	1201:
		_station.arrInfo[E_Language.Chinese]:="Z模组至取Uc位";
		IF M_ZTakeUc() THEN
			_station.iStepNext:=1301;
		END_IF
	1301:
		_station.arrInfo[E_Language.Chinese]:="夹紧气缸夹紧";
		IF G_arrFbCylinder[E_Cylinder.TakeUc1Clamp].M_WorkRequest() THEN
			_station.iStepNext:=1401;
		END_IF
	1401:
		_station.arrInfo[E_Language.Chinese]:="Z模组上升";
		IF M_ZHome() THEN
			_station.iStepNext:=1451;
		END_IF
	1451:
		_station.arrInfo[E_Language.Chinese]:="Y气缸至后位";
		G_arrFbCylinder[E_Cylinder.TakeUc1Y].M_WorkRequest();
		 _station.iStepNext:=1471;
	1471:
		_station.arrInfo[E_Language.Chinese]:="等待气缸到达安全点";
		IF GVL.I.bTakeUc1Y_Cyl_Safe OR GVL.I.bTakeUc1Y_Cyl_W THEN		
			_station.iStepNext:=1501;
		END_IF
	1501:
		_station.arrInfo[E_Language.Chinese]:="等待复位取Uc请求2";
		IF E_MachineType._311 = GVL_Data.stRecipe.eMachineType THEN
			IF NOT  GVL.stHandshake.bTakeUcToTakeUc_M_2 THEN
				GVL.stHandshake.bTakeUc_MToTakeUc_2:=FALSE;
				_station.iStepNext:=1601;
			END_IF
		ELSE
			IF NOT  GVL.stHandshake.bTakeUcToTakeUc_M THEN		
			  GVL.stHandshake.bTakeUc_MToTakeUc:=FALSE;			
				_station.iStepNext:=1551;
			END_IF	 
		END_IF 
	1551:
		_station.arrInfo[E_Language.Chinese]:="旋转气缸旋转";
		IF G_arrFbCylinder[E_Cylinder.TakeUc1Rotate].M_WorkRequest() AND G_arrFbCylinder[E_Cylinder.TakeUc1Y].M_WorkRequest() THEN
			_station.iStepNext:=1601;
		END_IF
	1601:
		_station.arrInfo[E_Language.Chinese]:="向下Uc皮带请求放料";
		GVL.stHandshake.bTakeUc_MToUnloadUcConveyor:=TRUE;
		IF GVL.stHandshake.bUnloadUcConveyorToTakeUc_M THEN
			_station.iStepNext:=1701;
		END_IF
	1701:
		_station.arrInfo[E_Language.Chinese]:="Z气缸下降放Uc";
		IF M_ZPlaceUc() THEN
			_station.iStepNext:=1801;
		END_IF
	1801:
		_station.arrInfo[E_Language.Chinese]:="夹紧气缸松开";
		IF G_arrFbCylinder[E_Cylinder.TakeUc1Clamp].M_HomeRequest() THEN
			_station.iStepNext:=1901;
		END_IF
	1901:
		_station.arrInfo[E_Language.Chinese]:="气缸上升";
		IF M_ZHome() THEN
			_station.iStepNext:=2001;
		END_IF
	2001:
	    _station.arrInfo[E_Language.Chinese]:="复位放料请求";
		GVL.stHandshake.bTakeUc_MToUnloadUcConveyor:=FALSE;
		IF NOT GVL.stHandshake.bUnloadUcConveyorToTakeUc_M THEN
		   	_station.iStepNext:=2101;
		END_IF
	2101:
		_station.arrInfo[E_Language.Chinese]:="旋转气缸复位";
		IF G_arrFbCylinder[E_Cylinder.TakeUc1Rotate].M_HomeRequest() THEN
			_station.iStepNext:=1101;
		END_IF
END_CASE
END_ACTION

ACTION A_Home:
CASE _station.iStepNow OF
	0:
		_station.arrInfo[E_Language.Chinese]:="等待初始化";
		_station.iStepNext:=SEL(_bEnable,1000,100);
	100:
		_station.arrInfo[E_Language.Chinese]:="夹紧气缸松开";
		IF G_arrFbCylinder[E_Cylinder.TakeUc1Clamp].M_HomeRequest() THEN
			_station.iStepNext:=200;
		END_IF
	200:
		_station.arrInfo[E_Language.Chinese]:="Z模组至待料位";
		IF M_ZHome() THEN
			_station.iStepNext:=300;
		END_IF		
	300:
		_station.arrInfo[E_Language.Chinese]:="旋转气缸复位";
		IF G_arrFbCylinder[E_Cylinder.TakeUc1Rotate].M_HomeRequest() THEN
			_station.iStepNext:=400;
		END_IF
	400:
		_station.arrInfo[E_Language.Chinese]:="Y气缸至后位";
	    IF G_arrFbCylinder[E_Cylinder.TakeUc1Y].M_WorkRequest() THEN
		    _station.iStepNext:=1000;
		END_IF
END_CASE
END_ACTION

METHOD M_ZHome : BOOL
VAR_INPUT
END_VAR
CASE GVL_Data.stRecipe.eMachineType OF
	E_MachineType._373:
	M_ZHome:=G_arrFbCylinder[E_Cylinder.TakeUc1Z1].M_HomeRequest();		
	ELSE
	M_ZHome:=G_arrFbCylinder[E_Cylinder.TakeUc1Z1].M_HomeRequest() AND G_arrFbCylinder[E_Cylinder.TakeUc1Z2].M_HomeRequest();
END_CASE
END_METHOD

METHOD M_ZPlaceUc : BOOL
VAR_INPUT
END_VAR
CASE GVL_Data.stRecipe.eMachineType OF
	E_MachineType._373:
	        M_ZPlaceUc:=G_arrFbCylinder[E_Cylinder.TakeUc1Z1].M_WorkRequest();
	E_MachineType._069: 
		    M_ZPlaceUc:=G_arrFbCylinder[E_Cylinder.TakeUc1Z1].M_WorkRequest() AND G_arrFbCylinder[E_Cylinder.TakeUc1Z2].M_WorkRequest();	
    E_MachineType._311:
			M_ZPlaceUc:=G_arrFbCylinder[E_Cylinder.TakeUc1Z1].M_WorkRequest();
	E_MachineType._367:
			M_ZPlaceUc:=G_arrFbCylinder[E_Cylinder.TakeUc1Z1].M_WorkRequest() AND G_arrFbCylinder[E_Cylinder.TakeUc1Z2].M_WorkRequest();
	E_MachineType._200:
	        M_ZPlaceUc:=G_arrFbCylinder[E_Cylinder.TakeUc1Z1].M_WorkRequest() AND G_arrFbCylinder[E_Cylinder.TakeUc1Z2].M_WorkRequest();
END_CASE
END_METHOD

METHOD M_ZTakeUc : BOOL
VAR_INPUT
END_VAR
CASE GVL_Data.stRecipe.eMachineType OF
	E_MachineType._373:
	    M_ZTakeUc:=G_arrFbCylinder[E_Cylinder.TakeUc1Z1].M_WorkRequest();	
	E_MachineType._069:
		    M_ZTakeUc:=G_arrFbCylinder[E_Cylinder.TakeUc1Z1].M_WorkRequest();
	E_MachineType._311:
	    M_ZTakeUc:=G_arrFbCylinder[E_Cylinder.TakeUc1Z1].M_WorkRequest() AND G_arrFbCylinder[E_Cylinder.TakeUc1Z2].M_WorkRequest();
	E_MachineType._367:
			M_ZTakeUc:=G_arrFbCylinder[E_Cylinder.TakeUc1Z2].M_WorkRequest();
	E_MachineType._200:
		   M_ZTakeUc:=G_arrFbCylinder[E_Cylinder.TakeUc1Z1].M_WorkRequest() AND G_arrFbCylinder[E_Cylinder.TakeUc1Z2].M_WorkRequest();
END_CASE
END_METHOD

END_PROGRAM

// ---- POUs/P_StationUnloadFrock.TcPOU
PROGRAM P_StationUnloadFrock
VAR
	_station:					REFERENCE TO ST_SystemStation;
	_bEnable: 					BOOL;
	
	_UnloadFrockCheck0FTrig:         Tc2_Standard.F_TRIG;
	
END_VAR

_station REF= G_arrStation[E_Station.UnloadFrock];
_station.arrName[E_Language.Chinese]:="下工装";
_station.arrName[E_Language.Vietnamese]:="Công cụ tiếp theo";
_bEnable:=NOT GVL.stSetting.arrStationShield[E_Station.UnloadFrock];
A_Auto();
A_Home();

_UnloadFrockCheck0FTrig(CLK:= GVL.I.bUnloadFrockCheck0, Q=> );

ACTION A_Auto:
CASE _station.iStepNow OF
	1000:
		_station.arrInfo[E_Language.Chinese]:="初始化完成等待启动";
		IF _bEnable THEN
			_station.iStepNext:=1101;
		END_IF
	1101:
		_station.arrInfo[E_Language.Chinese]:="判断是否有料";
		IF NOT GVL.I.bUnloadFrockCheck1 THEN
			_station.iStepNext:=1201;
		END_IF
	1201:
		_station.arrInfo[E_Language.Chinese]:="请求取Uc站放料";
		 GVL.stHandshake.bUnloadFrockToTakeUc:=TRUE;
		 IF  GVL.stHandshake.bTakeUcToUnloadFrock THEN
			 _station.iStepNext:=1301;
		 END_IF
	1301://安装了下工装站流入传感器但未移至阻挡气缸后侧启用此条
		_station.arrInfo[E_Language.Chinese]:="等待产品流入";
		GVL.stOverTime.bUnloadFrockCheck1:=TRUE; 
		IF NOT GVL.I.bTakeUcCheck1 AND GVL.I.bUnloadFrockCheck0 THEN
			GVL.stOverTime.bUnloadFrockCheck1:=FALSE; 
			_station.iStepNext:=1401;
		END_IF
		
(*	1301://安装了下工装站流入传感器并且移到了阻挡气缸后侧启用此条
		_station.arrInfo[E_Language.Chinese]:="等待产品从取UC站流出";
		GVL.stOverTime.bUnloadFrockCheck1:=TRUE; 
		IF NOT GVL.I.bTakeUcCheck1 THEN
			GVL.stOverTime.bUnloadFrockCheck1:=FALSE; 
			_station.iStepNext:=1311;
		END_IF		
	1311:		
		_station.arrInfo[E_Language.Chinese]:="产品从取UC站流出确认";
		IF _UnloadFrockCheck0FTrig.Q THEN
			_station.iStepNext:=1401;
		END_IF	*)	
	
	1401:
		_station.arrInfo[E_Language.Chinese]:="复位请求信号";
		 GVL.stHandshake.bUnloadFrockToTakeUc:=FALSE;
		 IF NOT GVL.stHandshake.bTakeUcToUnloadFrock THEN
			 _station.iStepNext:=1501;
		 END_IF
	1501:
		_station.arrInfo[E_Language.Chinese]:="等待产品到位";
		GVL.stOverTime.bUnloadFrockCheck1:=TRUE; 
		IF GVL.I.bUnloadFrockCheck1 THEN
			GVL.stOverTime.bUnloadFrockCheck1:=FALSE; 
			_station.iStepNext:=1601;
		END_IF
	1601:
		_station.arrInfo[E_Language.Chinese]:="顶升模组上升";
		IF M_LiftWork() THEN
			_station.iStepNext:=1651;
		END_IF
	1651:
		_station.arrInfo[E_Language.Chinese]:="向下工装线体请求放料";
		GVL.stHandshake.bUnloadFrockToUnloadFrock_L:=TRUE;
		IF  GVL.stHandshake.bUnloadFrock_LToUnloadFrock THEN
			_station.iStepNext:=1701;
		END_IF
	1701:
		_station.arrInfo[E_Language.Chinese]:="拨料气缸至后位";
		IF G_arrFbCylinder[E_Cylinder.UnloadFrockPush].M_WorkRequest()THEN
			_station.iStepNext:=1801;
		END_IF
	1801:
		_station.arrInfo[E_Language.Chinese]:="顶升模组下降 拨料气缸至前位";
		IF M_LiftHome() AND G_arrFbCylinder[E_Cylinder.UnloadFrockPush].M_HomeRequest() THEN
			_station.iStepNext:=2501;
		END_IF
	2501:
		_station.arrInfo[E_Language.Chinese]:="复位请求信号";
		GVL.stHandshake.bUnloadFrockToUnloadFrock_L:=FALSE;
		IF NOT GVL.stHandshake.bUnloadFrock_LToUnloadFrock THEN
			_station.iStepNext:=1101;
		END_IF
END_CASE
END_ACTION

ACTION A_Home:
CASE _station.iStepNow OF
	0:
		_station.arrInfo[E_Language.Chinese]:="等待初始化";
		_station.iStepNext:=SEL(_bEnable,1000,100);;
	100:
		_station.arrInfo[E_Language.Chinese]:="设备类型判断";
		_station.iStepNext:=200;
	200:
		_station.arrInfo[E_Language.Chinese]:="阻挡气缸伸出";
		CASE GVL_Data.stRecipe.eMachineType OF
			E_MachineType._200:
				IF G_arrFbCylinder[E_Cylinder.UnloadFrockPrevent].M_WorkRequest() THEN
					_station.iStepNext:=300;
				END_IF
			ELSE
				_station.iStepNext:=300;
		END_CASE
	300:
		_station.arrInfo[E_Language.Chinese]:="拨料气缸缩回";
		IF G_arrFbCylinder[E_Cylinder.UnloadFrockPush].M_HomeRequest() THEN
			_station.iStepNext:=350;
		END_IF		
	350:
		_station.arrInfo[E_Language.Chinese]:="顶升模组初始化";
		IF M_LiftInit() THEN
			_station.iStepNext:=400;
		END_IF
	400:		
		_station.arrInfo[E_Language.Chinese]:="顶升模组至下位";
		IF M_LiftHome() THEN
			_station.iStepNext:=1000;
		END_IF
END_CASE
END_ACTION

METHOD M_LiftHome : BOOL
VAR_INPUT
END_VAR
CASE GVL_Data.stRecipe.eMachineType OF
	E_MachineType._200:
		M_LiftHome:=G_arrFbCylinder[E_Cylinder.UnloadFrockLift].M_HomeRequest();
	ELSE
		M_LiftHome:=G_arrFbAxis[E_Axis.Z].M_MoveAbs(1);
END_CASE
END_METHOD

METHOD M_LiftInit : BOOL
VAR_INPUT
END_VAR
CASE GVL_Data.stRecipe.eMachineType OF
	E_MachineType._200:
		M_LiftInit:=G_arrFbCylinder[E_Cylinder.UnloadFrockLift].M_HomeRequest();
	ELSE
		M_LiftInit:=G_arrFbAxis[E_Axis.Z].M_Home();
END_CASE
END_METHOD

METHOD M_LiftWork : BOOL
VAR_INPUT
END_VAR
CASE GVL_Data.stRecipe.eMachineType OF
	E_MachineType._200:
		M_LiftWork:=G_arrFbCylinder[E_Cylinder.UnloadFrockLift].M_WorkRequest();
	ELSE
		M_LiftWork:=G_arrFbAxis[E_Axis.Z].M_MoveAbs(2);
END_CASE
END_METHOD

END_PROGRAM

// ---- POUs/P_StationUnloadFrock_L.TcPOU
PROGRAM P_StationUnloadFrock_L
VAR
	_station:					REFERENCE TO ST_SystemStation;
	_bEnable: 					BOOL;
	
	_bManual:                   BOOL;//  手动下料
END_VAR

_station REF= G_arrStation[E_Station.UnloadFrock_L];
_station.arrName[E_Language.Chinese]:="下工装线体";
_station.arrName[E_Language.Vietnamese]:="Thiết bị dây";
_bEnable:=NOT GVL.stSetting.arrStationShield[E_Station.UnloadFrock_L];

_bManual:=GVL.stSetting.bManualUnloadFrock;

A_Auto();
A_Home();

ACTION A_Auto:
CASE _station.iStepNow OF
	1000:
		_station.arrInfo[E_Language.Chinese]:="初始化完成等待启动";
		IF _bEnable THEN
			_station.iStepNext:=1101;
		END_IF
	1101:
		_station.arrInfo[E_Language.Chinese]:="判断是否有料";
		IF NOT GVL.I.bUnloadFrockConveyorCheck2 THEN
			_station.iStepNext:=1201;
		END_IF
	1201:
		_station.arrInfo[E_Language.Chinese]:="等待请求上料";
		IF GVL.stHandshake.bUnloadFrockToUnloadFrock_L THEN
			GVL.stHandshake.bUnloadFrock_LToUnloadFrock:=TRUE;
			_station.iStepNext:=1301;
		END_IF
	1301:
		_station.arrInfo[E_Language.Chinese]:="等待复位请求信号";
		IF NOT GVL.stHandshake.bUnloadFrockToUnloadFrock_L THEN
			GVL.stHandshake.bUnloadFrock_LToUnloadFrock:=FALSE;
			_station.iStepNext:=1401;
		END_IF
	1401:
		_station.arrInfo[E_Language.Chinese]:="等待产品到位";
		GVL.stOverTime.bUnloadFrockConveyorCheck2:=TRUE;
		IF GVL.I.bUnloadFrockConveyorCheck2 THEN
			GVL.stOverTime.bUnloadFrockConveyorCheck2:=FALSE;
			_station.iStepNext:=1451;
		END_IF
	1451:
		IF NOT _bManual  THEN
			_station.iStepNext:=1501;
			ELSE
			_station.iStepNext:=1101;
		END_IF
	1501:
		_station.arrInfo[E_Language.Chinese]:="升降气缸伸出";
		IF G_arrFbCylinder[E_Cylinder.UnloadFrockConveyorPrevent].M_WorkRequest() THEN
			_station.iStepNext:=1601;
		END_IF
	1601:
		_station.arrInfo[E_Language.Chinese]:="拨料气缸拨料";
		IF G_arrFbCylinder[E_Cylinder.UnloadFrockConveyorPush].M_WorkRequest() THEN
			_station.iStepNext:=1701;
		END_IF
	1701:
		_station.arrInfo[E_Language.Chinese]:="升降气缸缩回 拨料气缸缩回";
		IF  G_arrFbCylinder[E_Cylinder.UnloadFrockConveyorPush].M_HomeRequest() AND G_arrFbCylinder[E_Cylinder.UnloadFrockConveyorPrevent].M_HomeRequest() THEN
			_station.iStepNext:=1101;
		END_IF
END_CASE
END_ACTION

ACTION A_Home:
CASE _station.iStepNow OF
	0:
		_station.arrInfo[E_Language.Chinese]:="等待初始化";
		_station.iStepNext:=SEL(_bEnable,1000,100);
	100:
	    IF NOT _bManual  THEN
			_station.iStepNext:=200;
			ELSE
			_station.iStepNext:=1000;
		END_IF
	200:
		_station.arrInfo[E_Language.Chinese]:="升降气缸缩回";
		IF G_arrFbCylinder[E_Cylinder.UnloadFrockConveyorPrevent].M_HomeRequest() THEN
			_station.iStepNext:=300;
		END_IF
	300:
		_station.arrInfo[E_Language.Chinese]:="拨料气缸缩回";
		IF G_arrFbCylinder[E_Cylinder.UnloadFrockConveyorPush].M_HomeRequest() THEN
			_station.iStepNext:=1000;
		END_IF
END_CASE
END_ACTION

END_PROGRAM

// ---- POUs/P_StationUnloadUc_L.TcPOU
PROGRAM P_StationUnloadUc_L
VAR
	_station:					REFERENCE TO ST_SystemStation;
	_bEnable: 					BOOL;
	
	_ton:                       ARRAY [0..20] OF TON;;
	_frig:                      ARRAY [0..20] OF R_TRIG;
	_PreBelt:                   BOOL;
	
	_bManual:                   BOOL;//  手动下料
	
END_VAR

_station REF= G_arrStation[E_Station.UnloadUc_L];
_station.arrName[E_Language.Chinese]:="下Uc线体";
_station.arrName[E_Language.Vietnamese]:="Ống dẫn dưới UC";
_bEnable:=NOT GVL.stSetting.arrStationShield[E_Station.UnloadUc_L];

_bManual:=GVL.stSetting.bManualUnloadUc;

A_Auto();
A_Home();

ACTION A_Auto:
CASE _station.iStepNow OF
	1000:
		_station.arrInfo[E_Language.Chinese]:="初始化完成等待启动";
		IF _bEnable THEN
			_station.iStepNext:=1101;
		END_IF
	1101:
		_station.arrInfo[E_Language.Chinese]:="判断是否有料";
		IF NOT GVL.I.bUnloadUcCheck2 THEN
			_station.iStepNext:=SEL(GVL_Data.stRecipe.eMachineType=E_MachineType._200,1201,1111);
		END_IF
	1111:
		_station.arrInfo[E_Language.Chinese]:="顶升气缸伸出";
		IF G_arrFbCylinder[E_Cylinder.UnloadUcBeltLift].M_WorkRequest() THEN
			_station.iStepNext:=1201;
		END_IF
	1201:
		_station.arrInfo[E_Language.Chinese]:="等待请求上料";
		IF GVL.stHandshake.bTakeUc_MToUnloadUcConveyor THEN
			GVL.stHandshake.bUnloadUcConveyorToTakeUc_M:=TRUE;
			_station.iStepNext:=1301;
		END_IF
	1301:
		_station.arrInfo[E_Language.Chinese]:="等待复位请求信号";
		IF NOT GVL.stHandshake.bTakeUc_MToUnloadUcConveyor THEN
			GVL.stHandshake.bUnloadUcConveyorToTakeUc_M:=FALSE;
			_station.iStepNext:=1351;
		END_IF
	1351:
	     _station.arrInfo[E_Language.Chinese]:="开启下UC皮带线";
		 IF GVL.arrFbLine[E_LineAxis.UnloadUc].M_Jog(1) THEN
			IF  _bManual AND GVL.I.bUnloadUcCheck2 THEN
				GVL.arrFbLine[E_LineAxis.UnloadUc].M_Jog(0);
				_station.iStepNext:=1101;
			END_IF
			IF NOT _bManual THEN
				_station.iStepNext:=SEL(GVL_Data.stRecipe.eMachineType=E_MachineType._200,1501,1401);
			END_IF
		 END_IF
	1401:
		_station.arrInfo[E_Language.Chinese]:="等待产品到顶升位";
		GVL.stOverTime.bUnloadUcCheck1:=TRUE;
		IF gvl.I.bUnloadUcCheck1   THEN
			GVL.stOverTime.bUnloadUcCheck1:=FALSE;
			_station.iStepNext:=1451;
		END_IF
	1451:
		_station.arrInfo[E_Language.Chinese]:="翻转气缸动作";
		IF G_arrFbCylinder[E_Cylinder.UnloadUcBeltTipper].M_WorkRequest() THEN
			_station.iStepNext:=1471;
		END_IF
	1471:
		_station.arrInfo[E_Language.Chinese]:="顶升气缸缩回";
		IF G_arrFbCylinder[E_Cylinder.UnloadUcBeltLift].M_HomeRequest() THEN
			_station.iStepNext:=1501;
		END_IF 
	1501:
		_station.arrInfo[E_Language.Chinese]:="等待产品到拨料位";
		GVL.stOverTime.bUnloadUcCheck2 :=TRUE;
		IF GVL.I.bUnloadUcCheck2 THEN
			GVL.stOverTime.bUnloadUcCheck2 :=FALSE;
			GVL.arrFbLine[E_LineAxis.UnloadUc].M_Jog(0);
			_station.iStepNext:=1551;
		END_IF
	1551:
		_station.arrInfo[E_Language.Chinese]:="升降气缸伸出";
		IF G_arrFbCylinder[E_Cylinder.UnloadUcElevator].M_WorkRequest() THEN
			_station.iStepNext:=1601;
		END_IF
	1601:
		_station.arrInfo[E_Language.Chinese]:="拨料气缸拨料 翻转气缸复位";
		IF GVL_Data.stRecipe.eMachineType<>E_MachineType._200 THEN
			IF G_arrFbCylinder[E_Cylinder.UnloadUcConveyorPush].M_WorkRequest() THEN
				_station.iStepNext:=1701;
			END_IF
		ELSE
			IF G_arrFbCylinder[E_Cylinder.UnloadUcConveyorPush].M_WorkRequest() AND G_arrFbCylinder[E_Cylinder.UnloadUcBeltTipper].M_HomeRequest() THEN
				_station.iStepNext:=1701;
			END_IF
		END_IF
	1701:
		_station.arrInfo[E_Language.Chinese]:="升降气缸缩回 拨料气缸缩回";
		IF  G_arrFbCylinder[E_Cylinder.UnloadUcElevator].M_HomeRequest() AND G_arrFbCylinder[E_Cylinder.UnloadUcConveyorPush].M_HomeRequest() THEN
			_station.iStepNext:=1101;
		END_IF
END_CASE
END_ACTION

ACTION A_Home:
CASE _station.iStepNow OF
	0:
		_station.arrInfo[E_Language.Chinese]:="等待初始化";
		_station.iStepNext:=SEL(_bEnable AND NOT _bManual,1000,200);
	200:
		_station.arrInfo[E_Language.Chinese]:="升降气缸缩回";
		IF G_arrFbCylinder[E_Cylinder.UnloadUcElevator].M_HomeRequest() THEN
			_station.iStepNext:=300;
		END_IF
	300:
		_station.arrInfo[E_Language.Chinese]:="拨料气缸缩回";
		IF G_arrFbCylinder[E_Cylinder.UnloadUcConveyorPush].M_HomeRequest() THEN
			_station.iStepNext:=SEL(GVL_Data.stRecipe.eMachineType=E_MachineType._200,1000,500);
		END_IF
	500:
		_station.arrInfo[E_Language.Chinese]:="翻转气缸复位";
		IF G_arrFbCylinder[E_Cylinder.UnloadUcBeltTipper].M_HomeRequest() THEN
			_station.iStepNext:=600;
		END_IF
	600:
		_station.arrInfo[E_Language.Chinese]:="顶升气缸缩回";
		IF G_arrFbCylinder[E_Cylinder.UnloadUcBeltLift].M_HomeRequest() THEN
			_station.iStepNext:=1000;
		END_IF
END_CASE
END_ACTION

END_PROGRAM

// ---- POUs/P_StationLine1Load.TcPOU
PROGRAM P_StationLine1Load
VAR
	_station:					REFERENCE TO ST_SystemStation;
	_bEnable: 					BOOL;

END_VAR

_station REF= G_arrStation[E_Station.Line1Load];
_station.arrName[E_Language.Chinese]:="线条1上料站";
_station.arrName[E_Language.Vietnamese]:="Dòng trực tuyến";
_bEnable:= NOT GVL.stSetting.arrStationShield[E_Station.Line1Load] AND E_MachineType._367 <> GVL_Data.stRecipe.eMachineType;
GVL.stSetting.arrStationShield[E_Station.Line1Load]:=GVL.stSetting.bManualLoad;

A_Home();
A_Auto();

ACTION A_Auto:
CASE _station.iStepNow OF
	1000:
		_station.arrInfo[E_Language.Chinese]:="初始化完成等待启动";
		IF _bEnable  THEN
			_station.iStepNext:=1101;
		END_IF
	1101:
		_station.arrInfo[E_Language.Chinese]:="判断阻挡位是否有料";
		IF GVL.I.bAcquireCheck1 THEN
			_station.iStepNext:=1201;
		END_IF		
	1201:
		_station.arrInfo[E_Language.Chinese]:="接驳线前前阻挡气缸至工作位";	
		IF G_arrFbCylinder[E_Cylinder.AcquirePrevent2].M_WorkRequest() THEN 
			_station.iStepNext:=1301;
		END_IF
	1301:
		_station.arrInfo[E_Language.Chinese]:="接驳线请求接驳站收料";
		GVL.stHandshake.bLine1ToAcquire:=TRUE;
		IF GVL.stHandshake.bAcquireToLine1 THEN
			_station.iStepNext:=1401;
		END_IF
	1401:
		_station.arrInfo[E_Language.Chinese]:="前阻挡气缸缩回";
		IF G_arrFbCylinder[E_Cylinder.AcquirePrevent0].M_HomeRequest() THEN
			_station.iStepNext:=1501;
		END_IF
	1501:		
		_station.arrInfo[E_Language.Chinese]:="等待复位请求信号";
		IF NOT GVL.stHandshake.bAcquireToLine1 THEN
			GVL.stHandshake.bLine1ToAcquire:=FALSE;
			_station.iStepNext:=1601;
		END_IF
	1601:		
		_station.arrInfo[E_Language.Chinese]:="前阻挡气缸伸出";
		IF G_arrFbCylinder[E_Cylinder.AcquirePrevent0].M_WorkRequest() THEN
				_station.iStepNext:=1701;
		END_IF	
	1701:		
		_station.arrInfo[E_Language.Chinese]:="前前阻挡气缸缩回";
		IF G_arrFbCylinder[E_Cylinder.AcquirePrevent2].M_HomeRequest() THEN
			_station.iStepNext:=1101;
		END_IF
	
END_CASE
END_ACTION

ACTION A_Home:
CASE _station.iStepNow OF
	0:
		_station.arrInfo[E_Language.Chinese]:="等待初始化";
		_station.iStepNext:=SEL(_bEnable,1000,100);
	100:
		_station.arrInfo[E_Language.Chinese]:="阻挡气缸伸出";
		IF  G_arrFbCylinder[E_Cylinder.AcquirePrevent0].M_WorkRequest() THEN
			_station.iStepNext:=200;
		END_IF
	200:
		_station.arrInfo[E_Language.Chinese]:="分料气缸缩回";
		IF  G_arrFbCylinder[E_Cylinder.AcquirePrevent2].M_HomeRequest() THEN
			_station.iStepNext:=1000;
		END_IF
END_CASE
END_ACTION

END_PROGRAM

// ---- POUs/Device/FB_LineAxis.TcPOU
FUNCTION_BLOCK FB_LineAxis
VAR_INPUT
	Execute:				ST_TriggerMode;
	System:					REFERENCE TO ST_System;
END_VAR
VAR_OUTPUT
	Moving:					BOOL;
END_VAR
VAR
END_VAR

Moving:=FALSE;

IF System.stInput.bReset  THEN
	Moving:=FALSE;
	Execute.bAuto:=Execute.bManual:=FALSE;
END_IF

IF System.stMode.stDeviceRest.bAuto THEN
	Execute.bAuto:=FALSE;
END_IF
IF System.stMode.stDeviceRest.bManual THEN
	Execute.bManual:=FALSE;
END_IF

IF System.stMode.bAutoRunning THEN
	Moving:=Execute.bAuto;
END_IF
IF System.stMode.bManual THEN
	Moving:=Execute.bManual;
END_IF

METHOD M_Jog : BOOL
VAR_INPUT
	In:				INT;//0 停止 1正转
END_VAR
CASE In OF
	0:
		Execute.bAuto:=FALSE;
	1:
		Execute.bAuto:=TRUE;
END_CASE
M_Jog:=true;
END_METHOD

END_FUNCTION_BLOCK

// ---- GlobalTextList.TcGTLO
TEXTLIST GlobalTextList
  795 = '%'
  656 = '%0.1f'
  684 = '%0.2d'
  668 = '%0.2f'
  947 = '%d'
  268 = '%dms'
  858 = '%f'
  74 = '%s'
  761 = '1'
  1035 = '367机型' | Chinese: '367机型' | English: '367 Type' | Vietnamese: '367 Type'
  827 = 'Acquire'
  938 = 'Admin'
  67 = 'CT：%0.1f S'
  972 = 'Dismantling'
  258 = 'DryRun' | Chinese: '空跑' | English: 'DryRun' | Vietnamese: 'DryRun'
  238 = 'ioooo'
  355 = 'LED' | Chinese: '照明灯' | English: 'LED' | Vietnamese: 'LED'
  582 = 'Line0Buffer'
  240 = 'Line0BufferShield' | Chinese: '主流线分料屏蔽' | English: 'Line0BufferShield' | Vietnamese: 'Line1BufferShield'
  75 = 'LineAxis'
  978 = 'LUX' | Chinese: '立讯图标' | English: 'LUX' | Vietnamese: 'LUX'
  215 = 'ManualLoad' | Chinese: '手动上料' | English: 'ManualLoad' | Vietnamese: 'ManualLoad'
  475 = 'ManualUnloadFrock' | Chinese: '手动下工装' | English: 'ManualUnloadFrock' | Vietnamese: 'ManualUnloadFrock'
  177 = 'ManualUnloadUc' | Chinese: '手动下UC' | English: 'ManualUnloadUc' | Vietnamese: 'ManualUnloadUc'
  904 = 'None' | Chinese: '无' | English: 'None' | Vietnamese: 'None'
  186 = 'Operator'
  366 = 'Other'
  154 = 'Service'
  108 = 'UnloadForck' | Chinese: '下工装' | English: 'UnloadForck' | Vietnamese: 'UnloadForck'
  971 = 'UnloadUc' | Chinese: '下UC' | English: 'UnloadUc' | Vietnamese: 'UnloadUc'
  726 = 'Version:%s'
  288 = '上位' | Chinese: '上位' | English: 'Up Position' | Vietnamese: 'phán'
  486 = '上位:%dms' | Chinese: '上位:%dms' | English: 'Up Position:%dms' | Vietnamese: 'phán:%dms'
  370 = '下UC线体' | Chinese: '下UC线体' | English: 'UnloadUc' | Vietnamese: 'UnloadUc'
  109 = '下位' | Chinese: '下位' | English: 'Down Position' | Vietnamese: 'V? trí ti?p theo'
  409 = '下位:%dms' | Chinese: '下位:%dms' | English: 'Down Position:%dms' | Vietnamese: 'V? trí ti?p theo:%dms'
  286 = '下工装线体' | Chinese: '下工装线体' | English: 'UnloadForck' | Vietnamese: 'UnloadForck'
  646 = '不允许前站放料' | Chinese: '不允许前站放料' | English: 'StopFrontStation' | Vietnamese: 'StopFrontStation'
  399 = '主流线优先复位延时' | Chinese: '主流线优先置位延时' | English: 'Line0PriorityOnDelay' | Vietnamese: 'Line0PriorityOnDelay'
  738 = '主流线优先置位延时' | Chinese: '主流线优先复位延时' | English: 'Line0PriorityOffDelay' | Vietnamese: 'Line0PriorityOffDelay'
  758 = '主流线分料屏蔽' | Chinese: '主流线分料屏蔽' | English: 'Line0BufferShield' | Vietnamese: 'Line0BufferShield'
  687 = '主流线分料气缸缩回延时' | Chinese: '主流线分料气缸缩回延时' | English: 'Line0PartHomeDelay' | Vietnamese: 'Line0PartHomeDelay'
  750 = '伸出' | Chinese: '伸出' | English: 'Reach out' | Vietnamese: 'V??n ra'
  664 = '伸出:%dms' | Chinese: '伸出:%dms' | English: 'Reach out:%dms' | Vietnamese: 'V??n ra:%dms'
  716 = '伸出位' | Chinese: '伸出位' | English: 'Reach out' | Vietnamese: 'Thò tay ra'
  979 = '伸出位:%dms' | Chinese: '伸出位:%dms' | English: 'Reach out:%dms' | Vietnamese: 'Thò tay ra:%dms'
  554 = '保压解除功能屏蔽' | Chinese: '保压解除功能屏蔽' | English: 'OpenLockPressShield' | Vietnamese: 'OpenLockPressShield'
  477 = '共通' | Chinese: '共通' | English: 'Common' | Vietnamese: 'Common'
  941 = '初始位' | Chinese: '初始位' | English: 'Initial Position' | Vietnamese: 'Bit ban ??u'
  492 = '到位延迟' | Chinese: '到位延迟' | English: 'In delay' | Vietnamese: 'S? ch?m tr? t?i ch?'
  453 = '动位' | Chinese: '动位' | English: 'Action Position' | Vietnamese: 'Di chuy?n v? trí'
  45 = '动位:%dms' | Chinese: '动位:%dms' | English: 'Action Position:%dms' | Vietnamese: 'Di chuy?n v? trí:%dms'
  57 = '动作延迟' | Chinese: '动作延迟' | English: 'Action delay' | Vietnamese: 'S? trì ho?n hành ??ng'
  929 = '原位' | Chinese: '原位' | English: 'Home Position' | Vietnamese: '??'
  433 = '原位:%dms' | Chinese: '原位:%dms' | English: 'Home Position:%dms' | Vietnamese: '??:%dms'
  609 = '右位' | Chinese: '右位' | English: 'Right Position' | Vietnamese: 'Bên ph?i m?t'
  711 = '右位:%dms' | Chinese: '右位:%dms' | English: 'Right Position:%dms' | Vietnamese: 'Bên ph?i m?t:%dms'
  413 = '向上' | Chinese: '向上' | English: 'Up' | Vietnamese: '?i lên'
  498 = '向上:%dms' | Chinese: '向上:%dms' | English: 'Up:%dms' | Vietnamese: '?i lên:%dms'
  172 = '向下' | Chinese: '向下' | English: 'Down' | Vietnamese: 'Nhìn xu?ng'
  26 = '向下:%dms' | Chinese: '向下:%dms' | English: 'Down:%dms' | Vietnamese: 'Nhìn xu?ng:%dms'
  27 = '向右' | Chinese: '向右' | English: 'Right' | Vietnamese: 'Sang ph?i'
  151 = '向右:%dms' | Chinese: '向右:%dms' | English: 'Right:%dms' | Vietnamese: 'Sang ph?i:%dms'
  69 = '向左' | Chinese: '向左' | English: 'Left' | Vietnamese: 'Sang trái'
  849 = '向左:%dms' | Chinese: '向左:%dms' | English: 'Left:%dms' | Vietnamese: 'Sang trái:%dms'
  479 = '夹紧' | Chinese: '夹紧' | English: 'Clamp' | Vietnamese: 'K?p ch?t'
  504 = '夹紧:%dms' | Chinese: '夹紧:%dms' | English: 'Clamp:%dms' | Vietnamese: 'K?p ch?t:%dms'
  815 = '夹紧位' | Chinese: '夹紧位' | English: 'Clamp Position' | Vietnamese: 'k?p'
  925 = '夹紧位:%dms' | Chinese: '夹紧位:%dms' | English: 'Clamp Position:%dms' | Vietnamese: 'k?p:%dms'
  536 = '安全门屏蔽' | Chinese: '安全门屏蔽' | English: 'SafeDoorShield' | Vietnamese: 'SafeDoorShield'
  909 = '工作位' | Chinese: '工作位' | English: 'Work Position' | Vietnamese: 'V? trí làm vi?c'
  818 = '工装误合盖检测屏蔽' | Chinese: '工装误合盖检测屏蔽' | English: 'FrockCloseCheckShield' | Vietnamese: 'FrockCloseCheckShield'
  437 = '左位' | Chinese: '左位' | English: 'Left Position' | Vietnamese: 'M?t bên trái'
  165 = '左位:%dms' | Chinese: '左位:%dms' | English: 'Left Position:%dms' | Vietnamese: 'M?t bên trái:%dms'
  867 = '手动上料' | Chinese: '手动上料' | English: 'ManualLoad' | Vietnamese: 'bManualLoad'
  844 = '手动下UC' | Chinese: '手动下UC' | English: 'ManualUnloadUc' | Vietnamese: 'ManualUnloadUc'
  367 = '手动下工装' | Chinese: '手动下工装' | English: 'ManualUnloadFrock' | Vietnamese: 'ManualUnloadFrock'
  500 = '拆解线线体' | Chinese: '拆解线线体' | English: 'Dismantling' | Vietnamese: 'Dismantling'
  671 = '接驳站前线体' | Chinese: '接驳站前线体' | English: 'AcquireFront' | Vietnamese: 'AcquireFront'
  515 = '接驳站线体' | Chinese: '接驳站线体' | English: 'Acquire' | Vietnamese: 'Acquire'
  273 = '接驳线前前阻挡屏蔽' | Chinese: '接驳线前前阻挡屏蔽' | English: 'AcquirePrevent2Shield' | Vietnamese: 'AcquirePrevent2Shield'
  95 = '旋转站到位光电去抖动时间' | Chinese: '旋转站到位光电去抖动时间'
  885 = '旋转站到位检测光电去抖动时间'
  752 = '松开' | Chinese: '松开' | English: 'Loosen' | Vietnamese: 'Th? ra'
  628 = '松开:%dms' | Chinese: '松开:%dms' | English: 'Loosen:%dms' | Vietnamese: 'Th? ra:%dms'
  997 = '松开位' | Chinese: '松开位' | English: 'Loosen Position' | Vietnamese: 'N?i l?ng'
  836 = '松开位:%dms' | Chinese: '松开位:%dms' | English: 'Loosen Position:%dms' | Vietnamese: 'N?i l?ng:%dms'
  866 = '特瑞特'
  40 = '空跑' | Chinese: '空跑' | English: 'DryRun' | Vietnamese: 'DryRun'
  817 = '立讯图标' | Chinese: '立讯图标' | English: 'LIXUN' | Vietnamese: 'LIXUN'
  911 = '线体' | Chinese: '线体' | English: 'LineAxis' | Vietnamese: 'LineAxis'
  480 = '缩回' | Chinese: '缩回' | English: 'Retraction' | Vietnamese: 'Theo l?'
  875 = '缩回:%dms' | Chinese: '缩回:%dms' | English: 'Retraction:%dms' | Vietnamese: 'Theo l?:%dms'
  146 = '缩回位' | Chinese: '缩回位' | English: 'Retraction Position' | Vietnamese: 'Thu nh? các bit'
  589 = '缩回位:%dms' | Chinese: '缩回位:%dms' | English: 'Retraction Position:%dms' | Vietnamese: 'Thu nh? các bit:%dms'
  790 = '蜂鸣器屏蔽' | Chinese: '蜂鸣器屏蔽' | English: 'BuzzerShield' | Vietnamese: 'BuzzerShield'
  349 = '解锁站到位光电去抖动时间' | Chinese: '解锁站到位光电去抖动时间'
  824 = '计数清零' | Chinese: '计数清零' | English: 'Clear' | Vietnamese: 'Clear'
  830 = '输入' | Chinese: '输入' | English: 'Input' | Vietnamese: 'Nh?p vào'
  785 = '输出' | Chinese: '输出' | English: 'Output' | Vietnamese: '??u ra'
  872 = '远离' | Chinese: '远离' | English: 'Away from the screen' | Vietnamese: 'Tránh xa'
  195 = '远离:%dms' | Chinese: '远离:%dms' | English: 'Away from the screen:%dms' | Vietnamese: 'Tránh xa:%dms'
  449 = '远离位' | Chinese: '远离位' | English: 'Away from the screen' | Vietnamese: 'Tránh xa các bit'
  527 = '远离位:%dms' | Chinese: '远离位:%dms' | English: 'Away from the screen:%dms' | Vietnamese: 'Tránh xa các bit:%dms'
  14 = '远离屏幕' | Chinese: '远离屏幕' | English: 'Away from the screen' | Vietnamese: 'Tránh xa màn hình'
  587 = '释放' | Chinese: '释放' | English: 'Release' | Vietnamese: 'Gi?i phóng'
  719 = '靠近' | Chinese: '靠近' | English: 'Close to the screen' | Vietnamese: '??n g?n'
  569 = '靠近:%dms' | Chinese: '靠近:%dms' | English: 'Close to the screen:%dms' | Vietnamese: '??n g?n:%dms'
  786 = '靠近位' | Chinese: '靠近位' | English: 'Close to the screen' | Vietnamese: 'G?n v? trí'
  376 = '靠近位:%dms' | Chinese: '靠近位:%dms' | English: 'Close to the screen:%dms' | Vietnamese: 'G?n v? trí:%dms'
  549 = '靠近屏幕' | Chinese: '靠近屏幕' | English: 'Close to the screen' | Vietnamese: 'G?n màn hình'
  261 = '预留' | Chinese: '预留' | English: 'Reserved' | Vietnamese: 'Reserved'
END_TEXTLIST

// ---- VISUs/Ctrl/CtrlAxisInput.TcVIS
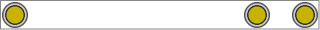
VISUALIZATION CtrlAxisInput  // 320x30
VAR_INPUT
	In:							UDINT;
END_VAR
    Lamp1 (0,0 30x30), variable: In.0, style: Lamp-Lamp1-Yellow
    Lamp1 (242,0 30x30), variable: In.2, style: Lamp-Lamp1-Yellow
    Lamp1 (290,0 30x30), variable: In.1, style: Lamp-Lamp1-Yellow
END_VISUALIZATION

// ---- VISUs/Ctrl/CtrlCylinder_Page.TcVIS
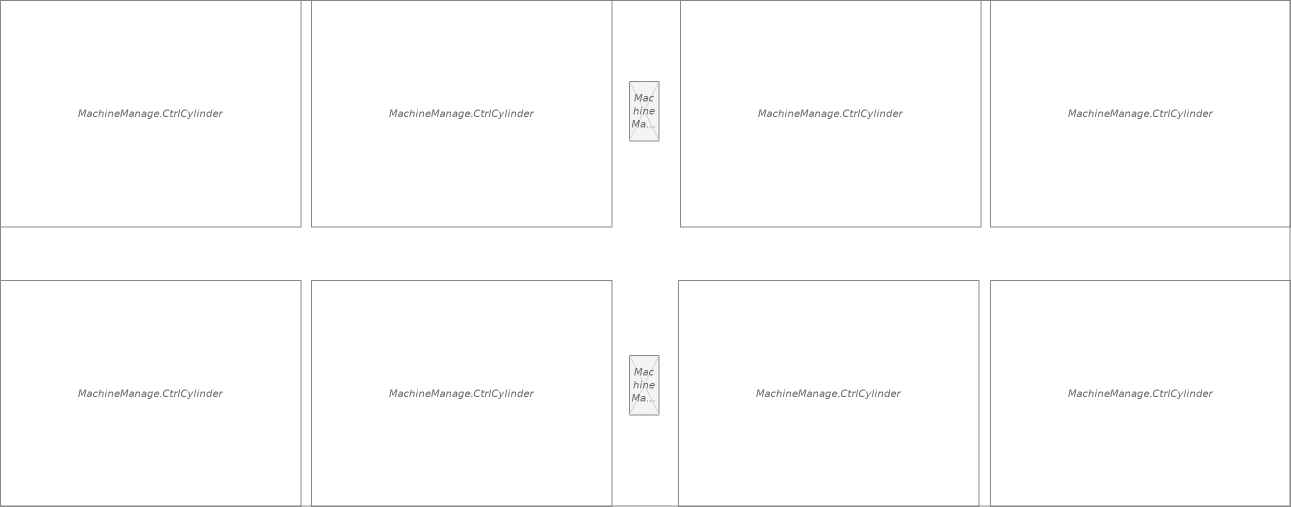
VISUALIZATION CtrlCylinder_Page  // 1291x507
VAR_INPUT
	System:				REFERENCE TO ST_System;
	Cylinder:			REFERENCE TO ARRAY[0..50] OF ST_Cylinder;
	CylinderData:		REFERENCE TO ARRAY[0..50] OF ST_CylinderData;
	Length:				INT;
END_VAR
VAR
	_i:					INT;
END_VAR
    Frame (0,0 301x227), invisible if: Length<=_i
        shows MachineManage.CtrlCylinder(System := System, Cylinder := Cylinder[_i], CylinderData := CylinderData[_i])
    Frame (311,0 301x227), invisible if: Length<=_i+1
        shows MachineManage.CtrlCylinder(System := System, Cylinder := Cylinder[_i+1], CylinderData := CylinderData[_i+1])
    Frame (0,280 301x227), invisible if: Length<=_i+2
        shows MachineManage.CtrlCylinder(System := System, Cylinder := Cylinder[_i+2], CylinderData := CylinderData[_i+2])
    Frame (311,280 301x227), invisible if: Length<=_i+3
        shows MachineManage.CtrlCylinder(System := System, Cylinder := Cylinder[_i+3], CylinderData := CylinderData[_i+3])
    Frame (680,0 301x227), invisible if: Length<=_i+4
        shows MachineManage.CtrlCylinder(System := System, Cylinder := Cylinder[_i+4], CylinderData := CylinderData[_i+4])
    Frame (678,280 301x227), invisible if: Length<=_i+6
        shows MachineManage.CtrlCylinder(System := System, Cylinder := Cylinder[_i+6], CylinderData := CylinderData[_i+6])
    Frame (990,0 301x227), invisible if: Length<=_i+5
        shows MachineManage.CtrlCylinder(System := System, Cylinder := Cylinder[_i+5], CylinderData := CylinderData[_i+5])
    Frame (990,280 301x227), invisible if: Length<=_i+7
        shows MachineManage.CtrlCylinder(System := System, Cylinder := Cylinder[_i+7], CylinderData := CylinderData[_i+7])
    Image (629,81 30x60), image: MachineManage.ImagePool.prev
        OnMouseDown: execute {
            IF _i-8>=0 THEN
            	_i:=_i-8;
            END_IF
        }
    Image (629,355 30x60), image: MachineManage.ImagePool.next
        OnMouseClick: execute {
            IF Length>_i+8 THEN
            	_i:=_i+8;
            END_IF
        }
END_VISUALIZATION

// ---- VISUs/Ctrl/CtrlLine.TcVIS
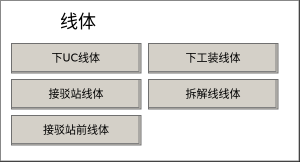
VISUALIZATION CtrlLine  // 300x162
    RoundedRectangle (0,0 300x162)
    Label (13,7 130x30), "线体"
    Button (11,43 130x30), "下UC线体"
        toggle GVL.arrFbLine[E_LineAxis.UnloadUc].Execute.bManual
    Button (148,43 130x30), "下工装线体"
        toggle GVL.arrFbLine[E_LineAxis.UnloadForck].Execute.bManual
    Button (11,79 130x30), "接驳站线体"
        toggle GVL.arrFbLine[E_LineAxis.Acquire].Execute.bManual
    Button (148,79 130x30), "拆解线线体"
        toggle GVL.arrFbLine[E_LineAxis.Dismantling].Execute.bManual
    Button (11,115 130x30), "接驳站前线体"
        toggle GVL.arrFbLine[E_LineAxis.AcquireFront].Execute.bManual
END_VISUALIZATION

// ---- VISUs/Ctrl/CtrlOutput.TcVIS
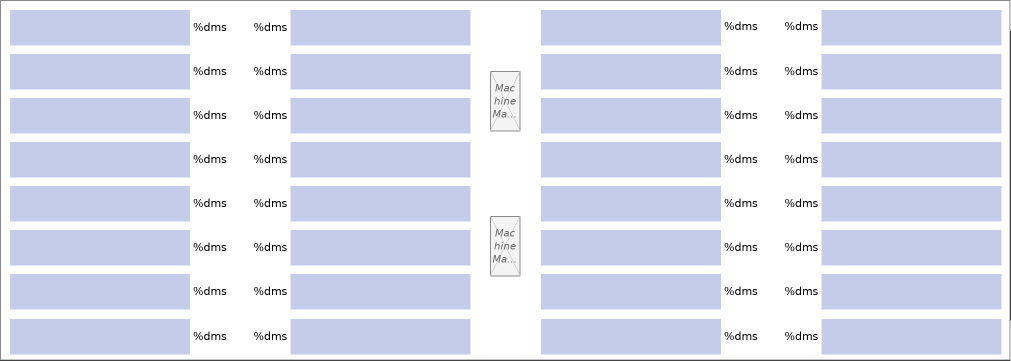
VISUALIZATION CtrlOutput  // 1011x361
VAR_INPUT
	In:						POINTER TO BOOL;
	SizeIn:					DINT;
	Enable:					BOOL;// 是否启用强制功能
	Ton:					POINTER TO UINT;// 延迟区域
	In_S:					POINTER TO BOOL;
END_VAR
VAR
	_pageCount:				INT;
	_index:					INT;
END_VAR
    RoundedRectangle (0,0 1010x115)
    RoundedRectangle (0,246 1010x115)
    Rectangle (0,52 1010x268)
    Line (1010,31) (1010,320)
    Line (0,33) (0,332)
    Image (490,71 30x60), image: MachineManage.ImagePool.prev
        OnMouseDown: execute {
            IF _index-32>=0 THEN
            	_index:=_index-32;
            END_IF
        }
    Image (490,216 30x60), image: MachineManage.ImagePool.next
        OnMouseClick: execute {
            IF SizeIn>_index+32 THEN
            	_index:=_index+32;
            END_IF
        }
    RoundedRectangle (10,10 180x35), colour toggle: In[_index], invisible if: SizeIn<=_index, input disabled if: In_S[_index], text list: 'OutputText', text index: _index
        OnMouseClick: execute {
            IF Enable AND SizeIn>_index THEN
            	In[_index]:=NOT In[_index];
            END_IF;
        }
    RoundedRectangle (10,54 180x35), colour toggle: In[1+_index], invisible if: SizeIn<= 1+_index, input disabled if: In_S[1+_index], text list: 'OutputText', text index: 1+_index
        OnMouseClick: execute {
            IF Enable AND SizeIn>_index+1 THEN
            	In[_index+1]:=NOT In[_index+1];
            END_IF;
        }
    RoundedRectangle (10,98 180x35), colour toggle: In[2+_index], invisible if: SizeIn<= 2+_index, input disabled if: In_S[2+_index], text list: 'OutputText', text index: 2+_index
        OnMouseClick: execute {
            IF Enable AND SizeIn>_index+2 THEN
            	In[_index+2]:=NOT In[_index+2];
            END_IF;
        }
    RoundedRectangle (10,142 180x35), colour toggle: In[3+_index], invisible if: SizeIn<=3+_index, input disabled if: In_S[3+_index], text list: 'OutputText', text index: 3+_index
        OnMouseClick: execute {
            IF Enable AND SizeIn>_index+3 THEN
            	In[_index+3]:=NOT In[_index+3];
            END_IF;
        }
    RoundedRectangle (10,186 180x35), colour toggle: In[_index+4], invisible if: SizeIn<=_index+4, input disabled if: In_S[_index+4], text list: 'OutputText', text index: _index+4
        OnMouseClick: execute {
            IF Enable AND SizeIn>_index+4 THEN
            	In[_index+4]:=NOT In[_index+4];
            END_IF;
        }
    RoundedRectangle (10,230 180x35), colour toggle: In[_index+5], invisible if: SizeIn<=_index+5, input disabled if: In_S[_index+5], text list: 'OutputText', text index: _index+5
        OnMouseClick: execute {
            IF Enable AND SizeIn>_index+5 THEN
            	In[_index+5]:=NOT In[_index+5];
            END_IF;
        }
    RoundedRectangle (10,274 180x35), colour toggle: In[_index+6], invisible if: SizeIn<=_index+6, input disabled if: In_S[_index+6], text list: 'OutputText', text index: _index+6
        OnMouseClick: execute {
            IF Enable AND SizeIn>_index+6 THEN
            	In[_index+6]:=NOT In[_index+6];
            END_IF;
        }
    RoundedRectangle (10,319 180x35), colour toggle: In[_index+7], invisible if: SizeIn<=_index+7, input disabled if: In_S[_index+7], text list: 'OutputText', text index: _index+7
        OnMouseClick: execute {
            IF Enable AND SizeIn>_index+7 THEN
            	In[_index+7]:=NOT In[_index+7];
            END_IF;
        }
    RoundedRectangle (290,10 180x35), colour toggle: In[_index+8], invisible if: SizeIn<=_index+8, input disabled if: In_S[_index+8], text list: 'OutputText', text index: _index+8
        OnMouseClick: execute {
            IF Enable AND SizeIn>_index+8 THEN
            	In[_index+8]:=NOT In[_index+8];
            END_IF;
        }
    RoundedRectangle (290,54 180x35), colour toggle: In[_index+9], invisible if: SizeIn<=_index+9, input disabled if: In_S[_index+9], text list: 'OutputText', text index: _index+9
        OnMouseClick: execute {
            IF Enable AND SizeIn>_index+9 THEN
            	In[_index+9]:=NOT In[_index+9];
            END_IF;
        }
    RoundedRectangle (290,98 180x35), colour toggle: In[_index+10], invisible if: SizeIn<=_index+10, input disabled if: In_S[_index+10], text list: 'OutputText', text index: _index+10
        OnMouseClick: execute {
            IF Enable AND SizeIn>_index+10 THEN
            	In[_index+10]:=NOT In[_index+10];
            END_IF;
        }
    RoundedRectangle (290,142 180x35), colour toggle: In[_index+11], invisible if: SizeIn<=_index+11, input disabled if: In_S[_index+11], text list: 'OutputText', text index: _index+11
        OnMouseClick: execute {
            IF Enable AND SizeIn>_index+11 THEN
            	In[_index+11]:=NOT In[_index+11];
            END_IF;
        }
    RoundedRectangle (290,186 180x35), colour toggle: In[_index+12], invisible if: SizeIn<=_index+12, input disabled if: In_S[_index+12], text list: 'OutputText', text index: _index+12
        OnMouseClick: execute {
            IF Enable AND SizeIn>_index+12 THEN
            	In[_index+12]:=NOT In[_index+12];
            END_IF;
        }
    RoundedRectangle (290,230 180x35), colour toggle: In[_index+13], invisible if: SizeIn<=_index+13, input disabled if: In_S[_index+13], text list: 'OutputText', text index: _index+13
        OnMouseClick: execute {
            IF Enable AND SizeIn>_index+13 THEN
            	In[_index+13]:=NOT In[_index+13];
            END_IF;
        }
    RoundedRectangle (290,274 180x35), colour toggle: In[_index+14], invisible if: SizeIn<=_index+14, input disabled if: In_S[_index+14], text list: 'OutputText', text index: _index+14
        OnMouseClick: execute {
            IF Enable AND SizeIn>_index+14 THEN
            	In[_index+14]:=NOT In[_index+14];
            END_IF;
        }
    RoundedRectangle (290,319 180x35), colour toggle: In[_index+15], invisible if: SizeIn<=_index+15, input disabled if: In_S[_index+15], text list: 'OutputText', text index: _index+15
        OnMouseClick: execute {
            IF Enable AND SizeIn>_index+15 THEN
            	In[_index+15]:=NOT In[_index+15];
            END_IF;
        }
    RoundedRectangle (541,10 180x35), colour toggle: In[_index+16], invisible if: SizeIn<=_index+16, input disabled if: In_S[_index+16], text list: 'OutputText', text index: _index+16
        OnMouseClick: execute {
            IF Enable AND SizeIn>_index+16 THEN
            	In[_index+16]:=NOT In[_index+16];
            END_IF;
        }
    RoundedRectangle (541,54 180x35), colour toggle: In[_index+17], invisible if: SizeIn<=_index+17, input disabled if: In_S[_index+17], text list: 'OutputText', text index: _index+17
        OnMouseClick: execute {
            IF Enable AND SizeIn>_index+17 THEN
            	In[_index+17]:=NOT In[_index+17];
            END_IF;
        }
    RoundedRectangle (541,98 180x35), colour toggle: In[_index+18], invisible if: SizeIn<=_index+18, input disabled if: In_S[_index+18], text list: 'OutputText', text index: _index+18
        OnMouseClick: execute {
            IF Enable AND SizeIn>_index+18 THEN
            	In[_index+18]:=NOT In[_index+18];
            END_IF;
        }
    RoundedRectangle (541,142 180x35), colour toggle: In[_index+19], invisible if: SizeIn<=_index+19, input disabled if: In_S[_index+19], text list: 'OutputText', text index: _index+19
        OnMouseClick: execute {
            IF Enable AND SizeIn>_index+19 THEN
            	In[_index+19]:=NOT In[_index+19];
            END_IF;
        }
    RoundedRectangle (541,186 180x35), colour toggle: In[_index+20], invisible if: SizeIn<=_index+20, input disabled if: In_S[_index+20], text list: 'OutputText', text index: _index+20
        OnMouseClick: execute {
            IF Enable AND SizeIn>_index+20 THEN
            	In[_index+20]:=NOT In[_index+20];
            END_IF;
        }
    RoundedRectangle (541,230 180x35), colour toggle: In[_index+21], invisible if: SizeIn<=_index+21, input disabled if: In_S[_index+21], text list: 'OutputText', text index: _index+21
        OnMouseClick: execute {
            IF Enable AND SizeIn>_index+21 THEN
            	In[_index+21]:=NOT In[_index+21];
            END_IF;
        }
    RoundedRectangle (541,274 180x35), colour toggle: In[_index+22], invisible if: SizeIn<=_index+22, input disabled if: In_S[_index+22], text list: 'OutputText', text index: _index+22
        OnMouseClick: execute {
            IF Enable AND SizeIn>_index+22 THEN
            	In[_index+22]:=NOT In[_index+22];
            END_IF;
        }
    RoundedRectangle (541,319 180x35), colour toggle: In[_index+23], invisible if: SizeIn<=_index+23, input disabled if: In_S[_index+23], text list: 'OutputText', text index: _index+23
        OnMouseClick: execute {
            IF Enable AND SizeIn>_index+23 THEN
            	In[_index+23]:=NOT In[_index+23];
            END_IF;
        }
    RoundedRectangle (821,10 180x35), colour toggle: In[_index+24], invisible if: SizeIn<=_index+24, input disabled if: In_S[_index+24], text list: 'OutputText', text index: _index+24
        OnMouseClick: execute {
            IF Enable AND SizeIn>_index+24 THEN
            	In[_index+24]:=NOT In[_index+24];
            END_IF;
        }
    RoundedRectangle (821,54 180x35), colour toggle: In[_index+25], invisible if: SizeIn<=_index+25, input disabled if: In_S[_index+25], text list: 'OutputText', text index: _index+25
        OnMouseClick: execute {
            IF Enable AND SizeIn>_index+25 THEN
            	In[_index+25]:=NOT In[_index+25];
            END_IF;
        }
    RoundedRectangle (821,98 180x35), colour toggle: In[_index+26], invisible if: SizeIn<=_index+26, input disabled if: In_S[_index+26], text list: 'OutputText', text index: _index+26
        OnMouseClick: execute {
            IF Enable AND SizeIn>_index+26 THEN
            	In[_index+26]:=NOT In[_index+26];
            END_IF;
        }
    RoundedRectangle (821,142 180x35), colour toggle: In[_index+27], invisible if: SizeIn<=_index+27, input disabled if: In_S[_index+27], text list: 'OutputText', text index: _index+27
        OnMouseClick: execute {
            IF Enable AND SizeIn>_index+27 THEN
            	In[_index+27]:=NOT In[_index+27];
            END_IF;
        }
    RoundedRectangle (821,186 180x35), colour toggle: In[_index+28], invisible if: SizeIn<=_index+28, input disabled if: In_S[_index+28], text list: 'OutputText', text index: _index+28
        OnMouseClick: execute {
            IF Enable AND SizeIn>_index+28 THEN
            	In[_index+28]:=NOT In[_index+28];
            END_IF;
        }
    RoundedRectangle (821,230 180x35), colour toggle: In[_index+29], invisible if: SizeIn<=_index+29, input disabled if: In_S[_index+29], text list: 'OutputText', text index: _index+29
        OnMouseClick: execute {
            IF Enable AND SizeIn>_index+29 THEN
            	In[_index+29]:=NOT In[_index+29];
            END_IF;
        }
    RoundedRectangle (821,274 180x35), colour toggle: In[_index+30], invisible if: SizeIn<=_index+30, input disabled if: In_S[_index+30], text list: 'OutputText', text index: _index+30
        OnMouseClick: execute {
            IF Enable AND SizeIn>_index+30 THEN
            	In[_index+30]:=NOT In[_index+30];
            END_IF;
        }
    RoundedRectangle (821,319 180x35), colour toggle: In[_index+31], invisible if: SizeIn<=_index+31, input disabled if: In_S[_index+31], text list: 'OutputText', text index: _index+31
        OnMouseClick: execute {
            IF Enable AND SizeIn>_index+31 THEN
            	In[_index+31]:=NOT In[_index+31];
            END_IF;
        }
    Rectangle (190,10 50x35), "%dms", text variable: Ton[_index], invisible if: SizeIn<=_index
        OnMouseClick: write the text variable via Default, min 0
    Rectangle (240,10 50x35), "%dms", text variable: Ton[_index+8], invisible if: SizeIn<=_index+8
        OnMouseClick: write the text variable via Default, min 0
    Rectangle (190,54 50x35), "%dms", text variable: Ton[_index+1], invisible if: SizeIn<=_index+1
        OnMouseClick: write the text variable via Default, min 0
    Rectangle (240,54 50x35), "%dms", text variable: Ton[_index+9], invisible if: SizeIn<=_index+9
        OnMouseClick: write the text variable via Default, min 0
    Rectangle (190,98 50x35), "%dms", text variable: Ton[_index+2], invisible if: SizeIn<=_index+2
        OnMouseClick: write the text variable via Default, min 0
    Rectangle (240,98 50x35), "%dms", text variable: Ton[_index+10], invisible if: SizeIn<=_index+10
        OnMouseClick: write the text variable via Default, min 0
    Rectangle (190,142 50x35), "%dms", text variable: Ton[_index+3], invisible if: SizeIn<=_index+3
        OnMouseClick: write the text variable via Default, min 0
    Rectangle (240,142 50x35), "%dms", text variable: Ton[_index+11], invisible if: SizeIn<=_index+11
        OnMouseClick: write the text variable via Default, min 0
    Rectangle (190,186 50x35), "%dms", text variable: Ton[_index+4], invisible if: SizeIn<=_index+4
        OnMouseClick: write the text variable via Default, min 0
    Rectangle (240,186 50x35), "%dms", text variable: Ton[_index+12], invisible if: SizeIn<=_index+12
        OnMouseClick: write the text variable via Default, min 0
    Rectangle (190,230 50x35), "%dms", text variable: Ton[_index+5], invisible if: SizeIn<=_index+5
        OnMouseClick: write the text variable via Default, min 0
    Rectangle (240,230 50x35), "%dms", text variable: Ton[_index+13], invisible if: SizeIn<=_index+13
        OnMouseClick: write the text variable via Default, min 0
    Rectangle (190,274 50x35), "%dms", text variable: Ton[_index+6], invisible if: SizeIn<=_index+6
        OnMouseClick: write the text variable via Default, min 0
    Rectangle (240,274 50x35), "%dms", text variable: Ton[_index+14], invisible if: SizeIn<=_index+14
        OnMouseClick: write the text variable via Default, min 0
    Rectangle (190,319 50x35), "%dms", text variable: Ton[_index+7], invisible if: SizeIn<=_index+7
        OnMouseClick: write the text variable via Default, min 0
    Rectangle (240,319 50x35), "%dms", text variable: Ton[_index+15], invisible if: SizeIn<=_index+15
        OnMouseClick: write the text variable via Default, min 0
    Rectangle (721,9 50x35), "%dms", text variable: Ton[_index+16], invisible if: SizeIn<=_index+16
        OnMouseClick: write the text variable via Default, min 0
    Rectangle (771,9 50x35), "%dms", text variable: Ton[_index+24], invisible if: SizeIn<=_index+24
        OnMouseClick: write the text variable via Default, min 0
    Rectangle (721,54 50x35), "%dms", text variable: Ton[_index+17], invisible if: SizeIn<=_index+17
        OnMouseClick: write the text variable via Default, min 0
    Rectangle (771,54 50x35), "%dms", text variable: Ton[_index+25], invisible if: SizeIn<=_index+25
        OnMouseClick: write the text variable via Default, min 0
    Rectangle (721,98 50x35), "%dms", text variable: Ton[_index+18], invisible if: SizeIn<=_index+18
        OnMouseClick: write the text variable via Default, min 0
    Rectangle (771,98 50x35), "%dms", text variable: Ton[_index+26], invisible if: SizeIn<=_index+26
        OnMouseClick: write the text variable via Default, min 0
    Rectangle (721,142 50x35), "%dms", text variable: Ton[_index+19], invisible if: SizeIn<=_index+19
        OnMouseClick: write the text variable via Default, min 0
    Rectangle (771,142 50x35), "%dms", text variable: Ton[_index+27], invisible if: SizeIn<=_index+27
        OnMouseClick: write the text variable via Default, min 0
    Rectangle (721,186 50x35), "%dms", text variable: Ton[_index+20], invisible if: SizeIn<=_index+20
        OnMouseClick: write the text variable via Default, min 0
    Rectangle (771,186 50x35), "%dms", text variable: Ton[_index+28], invisible if: SizeIn<=_index+28
        OnMouseClick: write the text variable via Default, min 0
    Rectangle (721,230 50x35), "%dms", text variable: Ton[_index+21], invisible if: SizeIn<=_index+21
        OnMouseClick: write the text variable via Default, min 0
    Rectangle (771,230 50x35), "%dms", text variable: Ton[_index+29], invisible if: SizeIn<=_index+29
        OnMouseClick: write the text variable via Default, min 0
    Rectangle (721,274 50x35), "%dms", text variable: Ton[_index+22], invisible if: SizeIn<=_index+22
        OnMouseClick: write the text variable via Default, min 0
    Rectangle (771,274 50x35), "%dms", text variable: Ton[_index+30], invisible if: SizeIn<=_index+30
        OnMouseClick: write the text variable via Default, min 0
    Rectangle (721,319 50x35), "%dms", text variable: Ton[_index+23], invisible if: SizeIn<=_index+23
        OnMouseClick: write the text variable via Default, min 0
    Rectangle (771,319 50x35), "%dms", text variable: Ton[_index+31], invisible if: SizeIn<=_index+31
        OnMouseClick: write the text variable via Default, min 0
END_VISUALIZATION

// ---- VISUs/Ctrl/Cyliner1.TcVIS
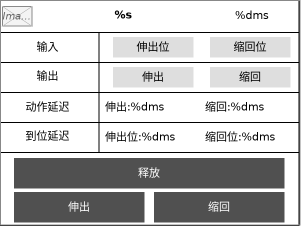
VISUALIZATION Cyliner1  // 301x226
VAR_INPUT
	System:							REFERENCE TO ST_System;
	Cylinder:						REFERENCE TO ST_Cylinder;
	CylinderData:					REFERENCE TO ST_CylinderData;
END_VAR
    RoundedRectangle (-1,111 300x115)
    RoundedRectangle (-1,0 300x115)
    Rectangle (-1,34 300x115)
    Line (-1,32) (299,32)
    Rectangle (34,3 179x24), "%s", text variable: Cylinder.arrInfo[System.stMode.eLanguage].sName, input disabled if: Cylinder.stLock.bShield
    Rectangle (217,3 70x25), "%dms", text variable: CylinderData.iAlarmTime, input disabled if: Cylinder.stLock.bShield
        OnMouseClick: write the text variable via VisuDialogs.Numpad
    Line (-1,62) (299,62)
    Line (-1,92) (299,92)
    Label (0,32 95x30), "输入"
    Label (0,61 95x30), "输出"
    Line (99,152) (99,32)
    RoundedRectangle (113,37 80x20), "伸出位", colour toggle: Cylinder.stInput.bWork, input disabled if: Cylinder.stLock.bShield
    RoundedRectangle (210,37 80x20), "缩回位", colour toggle: Cylinder.stInput.bHome, input disabled if: Cylinder.stLock.bShield
    RoundedRectangle (113,67 80x20), "伸出", colour toggle: Cylinder.stOutput.bWork, input disabled if: Cylinder.stLock.bShield
    RoundedRectangle (210,67 80x20), "缩回", colour toggle: Cylinder.stOutput.bHome, input disabled if: Cylinder.stLock.bShield
    RoundedRectangle (14,158 270x30), "释放", colour toggle: Cylinder.stLock.bOff OR Cylinder.stLock.bAll, input disabled if: Cylinder.stLock.bShield
        tap Cylinder.stControl.stOffRequest.bManual
    RoundedRectangle (14,192 130x30), "伸出", colour toggle: Cylinder.stLock.bWork OR Cylinder.stLock.bAll, input disabled if: Cylinder.stLock.bShield
        tap Cylinder.stControl.stWorkRequest.bManual
    RoundedRectangle (154,192 130x30), "缩回", colour toggle: Cylinder.stLock.bHome OR Cylinder.stLock.bAll, input disabled if: Cylinder.stLock.bShield
        tap Cylinder.stControl.stHomeRequest.bManual
    Line (299,154) (299,23)
    Line (-1,152) (-1,19)
    Image (2,6 30x20), image: ImagePool.Cylinder1
    Line (-1,122) (299,122)
    Line (-1,152) (299,152)
    Label (0,92 95x30), "动作延迟"
    Label (0,121 95x30), "到位延迟"
    RoundedRectangle (102,94 95x26), "伸出:%dms", text variable: CylinderData.iWorkRequestTime, input disabled if: Cylinder.stLock.bShield
        OnMouseClick: write the text variable via Default
    RoundedRectangle (202,94 95x26), "缩回:%dms", text variable: CylinderData.iHomeRequestTime, input disabled if: Cylinder.stLock.bShield
        OnMouseClick: write the text variable via Default
    RoundedRectangle (102,124 95x26), "伸出位:%dms", text variable: CylinderData.iWorkDone, input disabled if: Cylinder.stLock.bShield
        OnMouseClick: write the text variable via Default
    RoundedRectangle (202,124 95x26), "缩回位:%dms", text variable: CylinderData.iHomeDone, input disabled if: Cylinder.stLock.bShield
        OnMouseClick: write the text variable via Default
END_VISUALIZATION

// ---- VISUs/Ctrl/Cyliner1_1.TcVIS
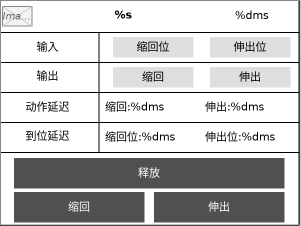
VISUALIZATION Cyliner1_1  // 301x226
VAR_INPUT
	System:							REFERENCE TO ST_System;
	Cylinder:						REFERENCE TO ST_Cylinder;
	CylinderData:					REFERENCE TO ST_CylinderData;
END_VAR
    RoundedRectangle (-1,111 300x115)
    RoundedRectangle (-1,0 300x115)
    Rectangle (-1,34 300x115)
    Line (-1,32) (299,32)
    Rectangle (34,3 179x24), "%s", text variable: Cylinder.arrInfo[System.stMode.eLanguage].sName, input disabled if: Cylinder.stLock.bShield
    Rectangle (217,3 70x25), "%dms", text variable: CylinderData.iAlarmTime, input disabled if: Cylinder.stLock.bShield
        OnMouseClick: write the text variable via VisuDialogs.Numpad
    Line (-1,62) (299,62)
    Line (-1,92) (299,92)
    Label (0,32 95x30), "输入"
    Label (0,61 95x30), "输出"
    Line (99,152) (99,32)
    RoundedRectangle (113,37 80x20), "缩回位", colour toggle: Cylinder.stInput.bWork, input disabled if: Cylinder.stLock.bShield
    RoundedRectangle (210,37 80x20), "伸出位", colour toggle: Cylinder.stInput.bHome, input disabled if: Cylinder.stLock.bShield
    RoundedRectangle (113,67 80x20), "缩回", colour toggle: Cylinder.stOutput.bWork, input disabled if: Cylinder.stLock.bShield
    RoundedRectangle (210,67 80x20), "伸出", colour toggle: Cylinder.stOutput.bHome, input disabled if: Cylinder.stLock.bShield
    RoundedRectangle (14,158 270x30), "释放", colour toggle: Cylinder.stLock.bOff OR Cylinder.stLock.bAll, input disabled if: Cylinder.stLock.bShield
        tap Cylinder.stControl.stOffRequest.bManual
    RoundedRectangle (14,192 130x30), "缩回", colour toggle: Cylinder.stLock.bWork OR Cylinder.stLock.bAll, input disabled if: Cylinder.stLock.bShield
        tap Cylinder.stControl.stWorkRequest.bManual
    RoundedRectangle (154,192 130x30), "伸出", colour toggle: Cylinder.stLock.bHome OR Cylinder.stLock.bAll, input disabled if: Cylinder.stLock.bShield
        tap Cylinder.stControl.stHomeRequest.bManual
    Line (299,154) (299,23)
    Line (-1,152) (-1,19)
    Image (2,6 30x20), image: ImagePool.Cylinder1
    Line (-1,122) (299,122)
    Line (-1,152) (299,152)
    Label (0,92 95x30), "动作延迟"
    Label (0,121 95x30), "到位延迟"
    RoundedRectangle (102,94 95x26), "缩回:%dms", text variable: CylinderData.iWorkRequestTime, input disabled if: Cylinder.stLock.bShield
        OnMouseClick: write the text variable via Default
    RoundedRectangle (202,94 95x26), "伸出:%dms", text variable: CylinderData.iHomeRequestTime, input disabled if: Cylinder.stLock.bShield
        OnMouseClick: write the text variable via Default
    RoundedRectangle (102,124 95x26), "缩回位:%dms", text variable: CylinderData.iWorkDone, input disabled if: Cylinder.stLock.bShield
        OnMouseClick: write the text variable via Default
    RoundedRectangle (202,124 95x26), "伸出位:%dms", text variable: CylinderData.iHomeDone, input disabled if: Cylinder.stLock.bShield
        OnMouseClick: write the text variable via Default
END_VISUALIZATION

// ---- VISUs/Ctrl/Cyliner2.TcVIS
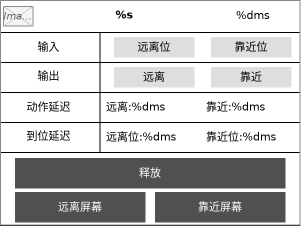
VISUALIZATION Cyliner2  // 301x226
VAR_INPUT
	System:							REFERENCE TO ST_System;
	Cylinder:						REFERENCE TO ST_Cylinder;
	CylinderData:					REFERENCE TO ST_CylinderData;
END_VAR
    RoundedRectangle (0,111 300x115)
    RoundedRectangle (0,0 300x115)
    Rectangle (0,34 300x115)
    Line (0,32) (300,32)
    Rectangle (35,3 179x24), "%s", text variable: Cylinder.arrInfo[System.stMode.eLanguage].sName, input disabled if: Cylinder.stLock.bShield
    Rectangle (218,3 70x25), "%dms", text variable: CylinderData.iAlarmTime, input disabled if: Cylinder.stLock.bShield
        OnMouseClick: write the text variable via VisuDialogs.Numpad
    Line (0,62) (300,62)
    Line (0,92) (300,92)
    Label (1,32 95x30), "输入"
    Label (1,61 95x30), "输出"
    Line (100,152) (100,32)
    RoundedRectangle (114,37 80x20), "远离位", colour toggle: Cylinder.stInput.bWork, input disabled if: Cylinder.stLock.bShield
    RoundedRectangle (211,37 80x20), "靠近位", colour toggle: Cylinder.stInput.bHome, input disabled if: Cylinder.stLock.bShield
    RoundedRectangle (114,67 80x20), "远离", colour toggle: Cylinder.stOutput.bWork, input disabled if: Cylinder.stLock.bShield
    RoundedRectangle (211,67 80x20), "靠近", colour toggle: Cylinder.stOutput.bHome, input disabled if: Cylinder.stLock.bShield
    RoundedRectangle (15,158 270x30), "释放", colour toggle: Cylinder.stLock.bOff OR Cylinder.stLock.bAll, input disabled if: Cylinder.stLock.bShield
        tap Cylinder.stControl.stOffRequest.bManual
    RoundedRectangle (15,192 130x30), "远离屏幕", colour toggle: Cylinder.stLock.bWork OR Cylinder.stLock.bAll, input disabled if: Cylinder.stLock.bShield
        tap Cylinder.stControl.stWorkRequest.bManual
    RoundedRectangle (155,192 130x30), "靠近屏幕", colour toggle: Cylinder.stLock.bHome OR Cylinder.stLock.bAll, input disabled if: Cylinder.stLock.bShield
        tap Cylinder.stControl.stHomeRequest.bManual
    Line (300,154) (300,23)
    Line (0,152) (0,19)
    Image (3,6 30x20), image: ImagePool.Cylinder1
    Line (0,122) (300,122)
    Line (0,152) (300,152)
    Label (1,92 95x30), "动作延迟"
    Label (1,121 95x30), "到位延迟"
    RoundedRectangle (103,94 95x26), "远离:%dms", text variable: CylinderData.iWorkRequestTime, input disabled if: Cylinder.stLock.bShield
        OnMouseClick: write the text variable via Default
    RoundedRectangle (203,94 95x26), "靠近:%dms", text variable: CylinderData.iHomeRequestTime, input disabled if: Cylinder.stLock.bShield
        OnMouseClick: write the text variable via Default
    RoundedRectangle (103,124 95x26), "远离位:%dms", text variable: CylinderData.iWorkDone, input disabled if: Cylinder.stLock.bShield
        OnMouseClick: write the text variable via Default
    RoundedRectangle (203,124 95x26), "靠近位:%dms", text variable: CylinderData.iHomeDone, input disabled if: Cylinder.stLock.bShield
        OnMouseClick: write the text variable via Default
END_VISUALIZATION

// ---- VISUs/Ctrl/Cyliner3.TcVIS
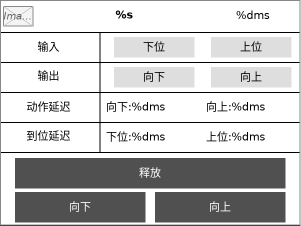
VISUALIZATION Cyliner3  // 301x226
VAR_INPUT
	System:							REFERENCE TO ST_System;
	Cylinder:						REFERENCE TO ST_Cylinder;
	CylinderData:					REFERENCE TO ST_CylinderData;
END_VAR
    RoundedRectangle (0,111 300x115)
    RoundedRectangle (0,0 300x115)
    Rectangle (0,34 300x115)
    Line (0,32) (300,32)
    Rectangle (35,3 179x24), "%s", text variable: Cylinder.arrInfo[System.stMode.eLanguage].sName, input disabled if: Cylinder.stLock.bShield
    Rectangle (218,3 70x25), "%dms", text variable: CylinderData.iAlarmTime, input disabled if: Cylinder.stLock.bShield
        OnMouseClick: write the text variable via VisuDialogs.Numpad
    Line (0,62) (300,62)
    Line (0,92) (300,92)
    Label (1,32 95x30), "输入"
    Label (1,61 95x30), "输出"
    Line (100,152) (100,32)
    RoundedRectangle (114,37 80x20), "下位", colour toggle: Cylinder.stInput.bWork, input disabled if: Cylinder.stLock.bShield
    RoundedRectangle (211,37 80x20), "上位", colour toggle: Cylinder.stInput.bHome, input disabled if: Cylinder.stLock.bShield
    RoundedRectangle (114,67 80x20), "向下", colour toggle: Cylinder.stOutput.bWork, input disabled if: Cylinder.stLock.bShield
    RoundedRectangle (211,67 80x20), "向上", colour toggle: Cylinder.stOutput.bHome, input disabled if: Cylinder.stLock.bShield
    RoundedRectangle (15,158 270x30), "释放", colour toggle: Cylinder.stLock.bOff OR Cylinder.stLock.bAll, input disabled if: Cylinder.stLock.bShield
        tap Cylinder.stControl.stOffRequest.bManual
    RoundedRectangle (15,192 130x30), "向下", colour toggle: Cylinder.stLock.bWork OR Cylinder.stLock.bAll, input disabled if: Cylinder.stLock.bShield
        tap Cylinder.stControl.stWorkRequest.bManual
    RoundedRectangle (155,192 130x30), "向上", colour toggle: Cylinder.stLock.bHome OR Cylinder.stLock.bAll, input disabled if: Cylinder.stLock.bShield
        tap Cylinder.stControl.stHomeRequest.bManual
    Line (300,154) (300,23)
    Line (0,152) (0,19)
    Image (3,6 30x20), image: ImagePool.Cylinder1
    Line (0,122) (300,122)
    Line (0,152) (300,152)
    Label (1,92 95x30), "动作延迟"
    Label (1,121 95x30), "到位延迟"
    RoundedRectangle (103,94 95x26), "向下:%dms", text variable: CylinderData.iWorkRequestTime, input disabled if: Cylinder.stLock.bShield
        OnMouseClick: write the text variable via Default
    RoundedRectangle (203,94 95x26), "向上:%dms", text variable: CylinderData.iHomeRequestTime, input disabled if: Cylinder.stLock.bShield
        OnMouseClick: write the text variable via Default
    RoundedRectangle (103,124 95x26), "下位:%dms", text variable: CylinderData.iWorkDone, input disabled if: Cylinder.stLock.bShield
        OnMouseClick: write the text variable via Default
    RoundedRectangle (203,124 95x26), "上位:%dms", text variable: CylinderData.iHomeDone, input disabled if: Cylinder.stLock.bShield
        OnMouseClick: write the text variable via Default
END_VISUALIZATION

// ---- VISUs/Ctrl/Cyliner4.TcVIS
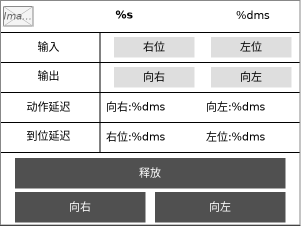
VISUALIZATION Cyliner4  // 301x226
VAR_INPUT
	System:							REFERENCE TO ST_System;
	Cylinder:						REFERENCE TO ST_Cylinder;
	CylinderData:					REFERENCE TO ST_CylinderData;
END_VAR
    RoundedRectangle (0,111 300x115)
    RoundedRectangle (0,0 300x115)
    Rectangle (0,34 300x115)
    Line (0,32) (300,32)
    Rectangle (35,3 179x24), "%s", text variable: Cylinder.arrInfo[System.stMode.eLanguage].sName, input disabled if: Cylinder.stLock.bShield
    Rectangle (218,3 70x25), "%dms", text variable: CylinderData.iAlarmTime, input disabled if: Cylinder.stLock.bShield
        OnMouseClick: write the text variable via VisuDialogs.Numpad
    Line (0,62) (300,62)
    Line (0,92) (300,92)
    Label (1,32 95x30), "输入"
    Label (1,61 95x30), "输出"
    Line (100,152) (100,32)
    RoundedRectangle (114,37 80x20), "右位", colour toggle: Cylinder.stInput.bWork, input disabled if: Cylinder.stLock.bShield
    RoundedRectangle (211,37 80x20), "左位", colour toggle: Cylinder.stInput.bHome, input disabled if: Cylinder.stLock.bShield
    RoundedRectangle (114,67 80x20), "向右", colour toggle: Cylinder.stOutput.bWork, input disabled if: Cylinder.stLock.bShield
    RoundedRectangle (211,67 80x20), "向左", colour toggle: Cylinder.stOutput.bHome, input disabled if: Cylinder.stLock.bShield
    RoundedRectangle (15,158 270x30), "释放", colour toggle: Cylinder.stLock.bOff OR Cylinder.stLock.bAll, input disabled if: Cylinder.stLock.bShield
        tap Cylinder.stControl.stOffRequest.bManual
    RoundedRectangle (15,192 130x30), "向右", colour toggle: Cylinder.stLock.bWork OR Cylinder.stLock.bAll, input disabled if: Cylinder.stLock.bShield
        tap Cylinder.stControl.stWorkRequest.bManual
    RoundedRectangle (155,192 130x30), "向左", colour toggle: Cylinder.stLock.bHome OR Cylinder.stLock.bAll, input disabled if: Cylinder.stLock.bShield
        tap Cylinder.stControl.stHomeRequest.bManual
    Line (300,154) (300,23)
    Line (0,152) (0,19)
    Image (3,6 30x20), image: ImagePool.Cylinder1
    Line (0,122) (300,122)
    Line (0,152) (300,152)
    Label (1,92 95x30), "动作延迟"
    Label (1,121 95x30), "到位延迟"
    RoundedRectangle (103,94 95x26), "向右:%dms", text variable: CylinderData.iWorkRequestTime, input disabled if: Cylinder.stLock.bShield
        OnMouseClick: write the text variable via Default
    RoundedRectangle (203,94 95x26), "向左:%dms", text variable: CylinderData.iHomeRequestTime, input disabled if: Cylinder.stLock.bShield
        OnMouseClick: write the text variable via Default
    RoundedRectangle (103,124 95x26), "右位:%dms", text variable: CylinderData.iWorkDone, input disabled if: Cylinder.stLock.bShield
        OnMouseClick: write the text variable via Default
    RoundedRectangle (203,124 95x26), "左位:%dms", text variable: CylinderData.iHomeDone, input disabled if: Cylinder.stLock.bShield
        OnMouseClick: write the text variable via Default
END_VISUALIZATION

// ---- VISUs/Ctrl/Cyliner4_1.TcVIS
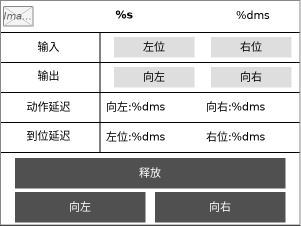
VISUALIZATION Cyliner4_1  // 301x226
VAR_INPUT
	System:							REFERENCE TO ST_System;
	Cylinder:						REFERENCE TO ST_Cylinder;
	CylinderData:					REFERENCE TO ST_CylinderData;
END_VAR
    RoundedRectangle (0,111 300x115)
    RoundedRectangle (0,0 300x115)
    Rectangle (0,34 300x115)
    Line (0,32) (300,32)
    Rectangle (35,3 179x24), "%s", text variable: Cylinder.arrInfo[System.stMode.eLanguage].sName, input disabled if: Cylinder.stLock.bShield
    Rectangle (218,3 70x25), "%dms", text variable: CylinderData.iAlarmTime, input disabled if: Cylinder.stLock.bShield
        OnMouseClick: write the text variable via VisuDialogs.Numpad
    Line (0,62) (300,62)
    Line (0,92) (300,92)
    Label (1,32 95x30), "输入"
    Label (1,61 95x30), "输出"
    Line (100,152) (100,32)
    RoundedRectangle (114,37 80x20), "左位", colour toggle: Cylinder.stInput.bWork, input disabled if: Cylinder.stLock.bShield
    RoundedRectangle (211,37 80x20), "右位", colour toggle: Cylinder.stInput.bHome, input disabled if: Cylinder.stLock.bShield
    RoundedRectangle (114,67 80x20), "向左", colour toggle: Cylinder.stOutput.bWork, input disabled if: Cylinder.stLock.bShield
    RoundedRectangle (211,67 80x20), "向右", colour toggle: Cylinder.stOutput.bHome, input disabled if: Cylinder.stLock.bShield
    RoundedRectangle (15,158 270x30), "释放", colour toggle: Cylinder.stLock.bOff OR Cylinder.stLock.bAll, input disabled if: Cylinder.stLock.bShield
        tap Cylinder.stControl.stOffRequest.bManual
    RoundedRectangle (15,192 130x30), "向左", colour toggle: Cylinder.stLock.bWork OR Cylinder.stLock.bAll, input disabled if: Cylinder.stLock.bShield
        tap Cylinder.stControl.stWorkRequest.bManual
    RoundedRectangle (155,192 130x30), "向右", colour toggle: Cylinder.stLock.bHome OR Cylinder.stLock.bAll, input disabled if: Cylinder.stLock.bShield
        tap Cylinder.stControl.stHomeRequest.bManual
    Line (300,154) (300,23)
    Line (0,152) (0,19)
    Image (3,6 30x20), image: ImagePool.Cylinder1
    Line (0,122) (300,122)
    Line (0,152) (300,152)
    Label (1,92 95x30), "动作延迟"
    Label (1,121 95x30), "到位延迟"
    RoundedRectangle (103,94 95x26), "向左:%dms", text variable: CylinderData.iWorkRequestTime, input disabled if: Cylinder.stLock.bShield
        OnMouseClick: write the text variable via Default
    RoundedRectangle (203,94 95x26), "向右:%dms", text variable: CylinderData.iHomeRequestTime, input disabled if: Cylinder.stLock.bShield
        OnMouseClick: write the text variable via Default
    RoundedRectangle (103,124 95x26), "左位:%dms", text variable: CylinderData.iWorkDone, input disabled if: Cylinder.stLock.bShield
        OnMouseClick: write the text variable via Default
    RoundedRectangle (203,124 95x26), "右位:%dms", text variable: CylinderData.iHomeDone, input disabled if: Cylinder.stLock.bShield
        OnMouseClick: write the text variable via Default
END_VISUALIZATION

// ---- VISUs/Ctrl/Cyliner5.TcVIS
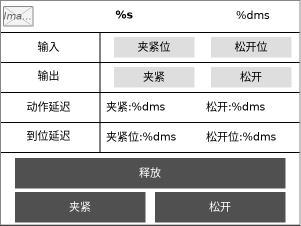
VISUALIZATION Cyliner5  // 301x226
VAR_INPUT
	System:							REFERENCE TO ST_System;
	Cylinder:						REFERENCE TO ST_Cylinder;
	CylinderData:					REFERENCE TO ST_CylinderData;
END_VAR
    RoundedRectangle (0,111 300x115)
    RoundedRectangle (0,0 300x115)
    Rectangle (0,34 300x115)
    Line (0,32) (300,32)
    Rectangle (35,3 179x24), "%s", text variable: Cylinder.arrInfo[System.stMode.eLanguage].sName, input disabled if: Cylinder.stLock.bShield
    Rectangle (218,3 70x25), "%dms", text variable: CylinderData.iAlarmTime, input disabled if: Cylinder.stLock.bShield
        OnMouseClick: write the text variable via VisuDialogs.Numpad
    Line (0,62) (300,62)
    Line (0,92) (300,92)
    Label (1,32 95x30), "输入"
    Label (1,61 95x30), "输出"
    Line (100,152) (100,32)
    RoundedRectangle (114,37 80x20), "夹紧位", colour toggle: Cylinder.stInput.bWork, input disabled if: Cylinder.stLock.bShield
    RoundedRectangle (211,37 80x20), "松开位", colour toggle: Cylinder.stInput.bHome, input disabled if: Cylinder.stLock.bShield
    RoundedRectangle (114,67 80x20), "夹紧", colour toggle: Cylinder.stOutput.bWork, input disabled if: Cylinder.stLock.bShield
    RoundedRectangle (211,67 80x20), "松开", colour toggle: Cylinder.stOutput.bHome, input disabled if: Cylinder.stLock.bShield
    RoundedRectangle (15,158 270x30), "释放", colour toggle: Cylinder.stLock.bOff OR Cylinder.stLock.bAll, input disabled if: Cylinder.stLock.bShield
        tap Cylinder.stControl.stOffRequest.bManual
    RoundedRectangle (15,192 130x30), "夹紧", colour toggle: Cylinder.stLock.bWork OR Cylinder.stLock.bAll, input disabled if: Cylinder.stLock.bShield
        tap Cylinder.stControl.stWorkRequest.bManual
    RoundedRectangle (155,192 130x30), "松开", colour toggle: Cylinder.stLock.bHome OR Cylinder.stLock.bAll, input disabled if: Cylinder.stLock.bShield
        tap Cylinder.stControl.stHomeRequest.bManual
    Line (300,154) (300,23)
    Line (0,152) (0,19)
    Image (3,6 30x20), image: ImagePool.Cylinder1
    Line (0,122) (300,122)
    Line (0,152) (300,152)
    Label (1,92 95x30), "动作延迟"
    Label (1,121 95x30), "到位延迟"
    RoundedRectangle (103,94 95x26), "夹紧:%dms", text variable: CylinderData.iWorkRequestTime, input disabled if: Cylinder.stLock.bShield
        OnMouseClick: write the text variable via Default
    RoundedRectangle (203,94 95x26), "松开:%dms", text variable: CylinderData.iHomeRequestTime, input disabled if: Cylinder.stLock.bShield
        OnMouseClick: write the text variable via Default
    RoundedRectangle (103,124 95x26), "夹紧位:%dms", text variable: CylinderData.iWorkDone, input disabled if: Cylinder.stLock.bShield
        OnMouseClick: write the text variable via Default
    RoundedRectangle (203,124 95x26), "松开位:%dms", text variable: CylinderData.iHomeDone, input disabled if: Cylinder.stLock.bShield
        OnMouseClick: write the text variable via Default
END_VISUALIZATION

// ---- VISUs/Ctrl/FrameMain.TcVIS
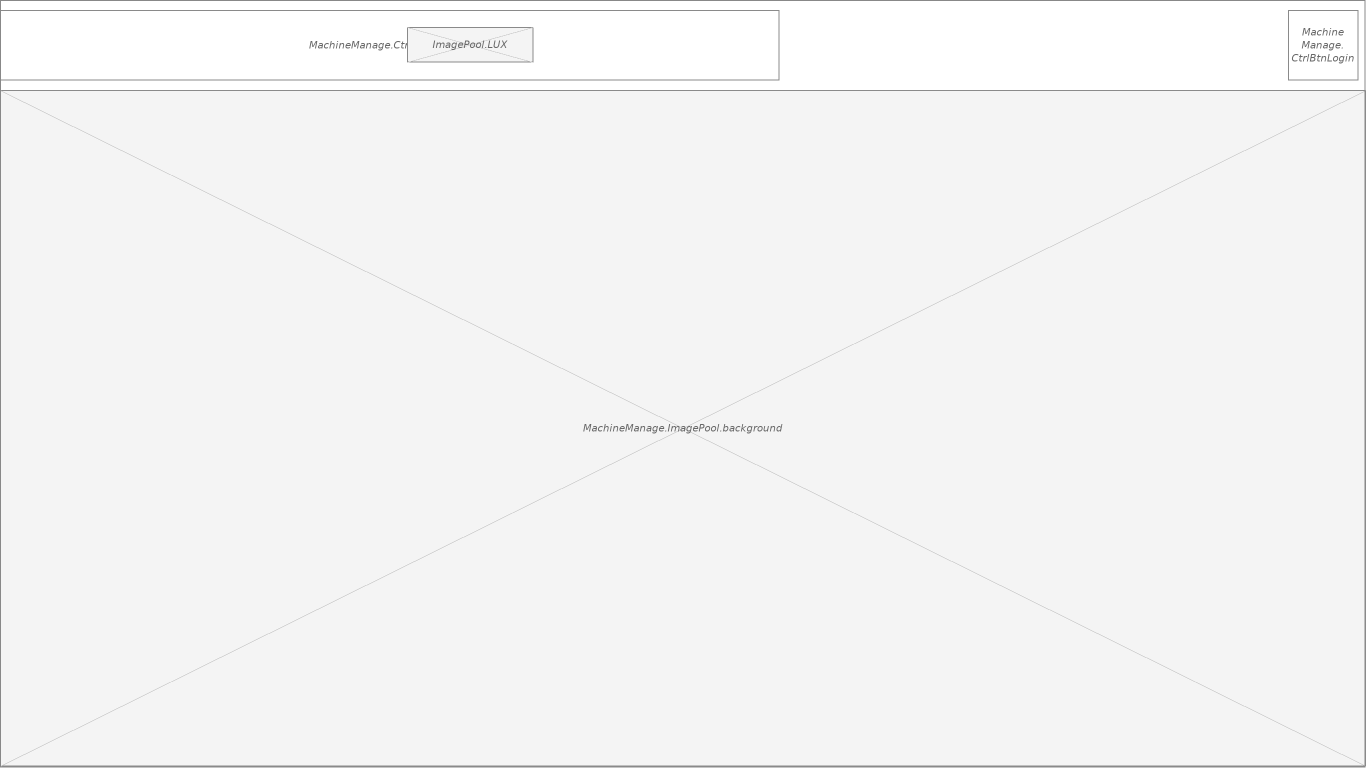
VISUALIZATION FrameMain  // 1366x768
    Frame (0,10 779x70)
        shows MachineManage.CtrlPageSwitch(System := G_stSystem)
    Image (0,90 1366x676), image: MachineManage.ImagePool.background
    Frame (1288,10 70x70)
        shows MachineManage.CtrlBtnLogin()
    Rectangle (414,30 113x32), "Goertek"
    Image (407,27 126x35), invisible if: NOT GVL_Data.stRecipe.bLuxshardict, image: ImagePool.LUX
END_VISUALIZATION

// ---- VISUs/Ctrl/CtrlPageSetting.TcVIS
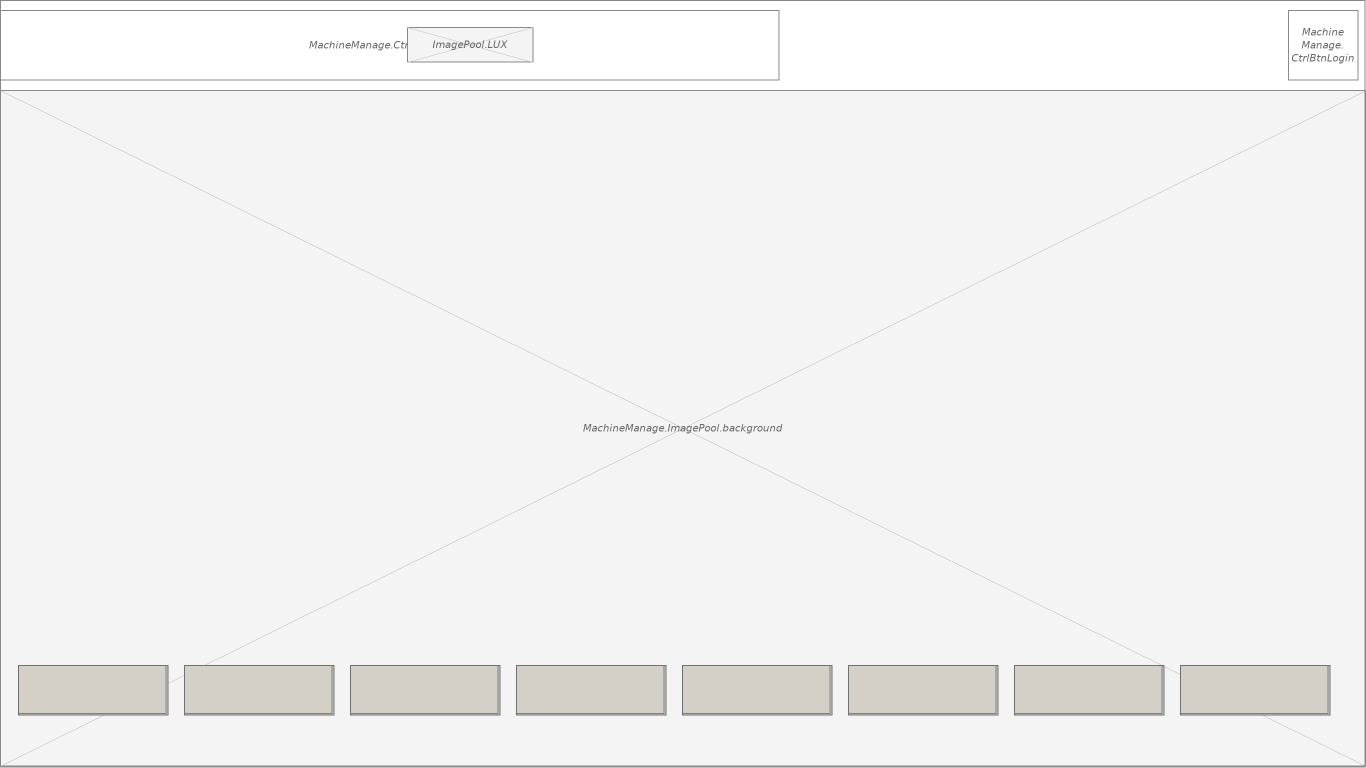
VISUALIZATION CtrlPageSetting  // 1366x768
    Frame (0,0 1366x768)
        shows FrameMain()
    Button (18,665 150x50), text list: 'StationName', text index: 0
        OnMouseClick: change screen: PageSetting_AcquireLoad
    Button (184,665 150x50), text list: 'StationName', text index: 1
        OnMouseClick: change screen: PageSetting_Steering
    Button (350,665 150x50), text list: 'StationName', text index: 2
        OnMouseClick: change screen: PageSetting_OpenLock
    Button (516,665 150x50), text list: 'StationName', text index: 3
        OnMouseClick: change screen: PageSetting_TakeUc
    Button (682,665 150x50), text list: 'StationName', text index: 4
        OnMouseClick: change screen: PageSetting_TakeUc_M
    Button (848,665 150x50), text list: 'StationName', text index: 5
        OnMouseClick: change screen: PageSetting_UnloadFrock
    Button (1014,665 150x50), text list: 'StationName', text index: 6
        OnMouseClick: change screen: PageSetting_Unload_L
    Button (1180,665 150x50), text list: 'StationName', text index: 7
        OnMouseClick: change screen: PageSetting_Other
END_VISUALIZATION

// ---- VISUs/PageData.TcVIS
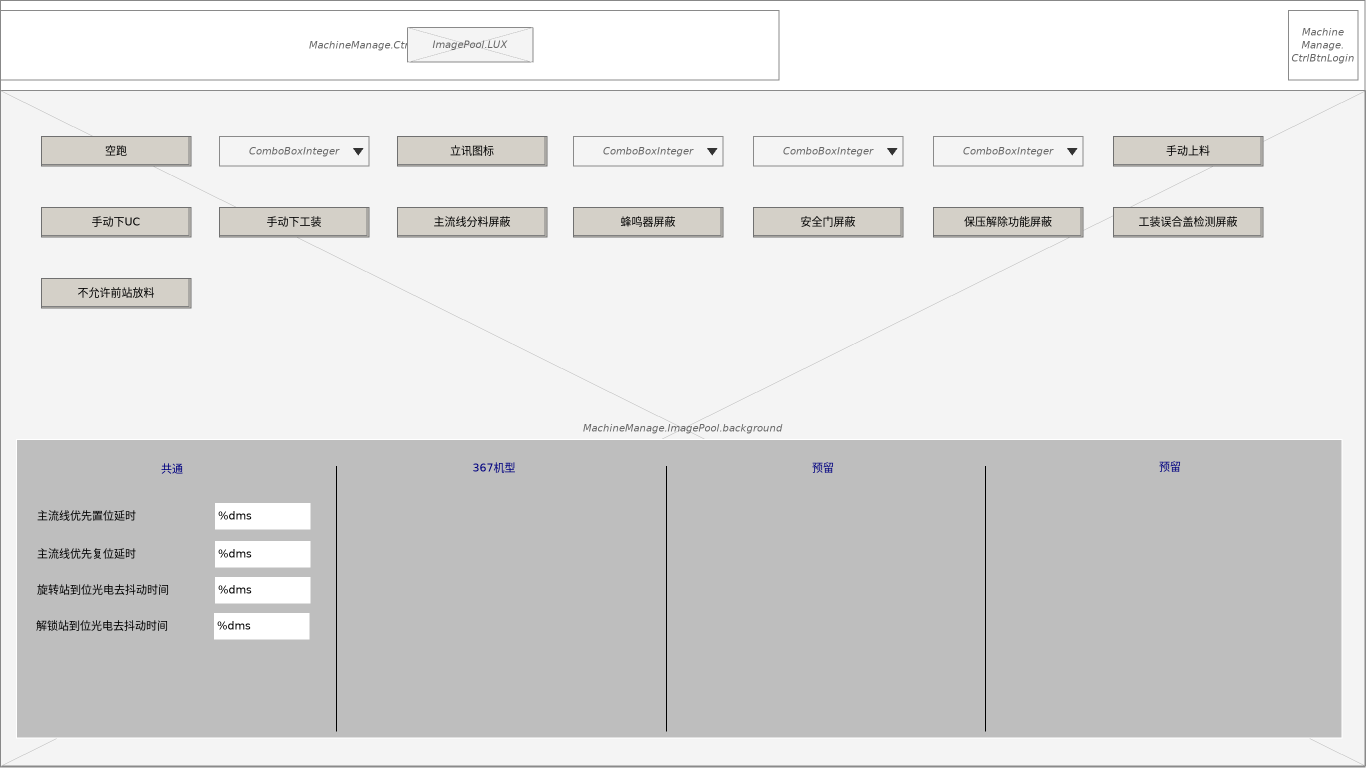
VISUALIZATION PageData  // 1366x768
    Frame (0,0 1366x768)
        shows FrameMain()
    Rectangle (16,439 1326x299)
    Button (41,136 150x30), "空跑"
        toggle GVL.stSetting.bDryRun
    ComboBoxInteger (219,136 150x30), variable: GVL_Data.stRecipe.eMachineType, text list: 'MachineType'
    Button (397,136 150x30), "立讯图标"
        toggle GVL_Data.stRecipe.bLuxshardict
    ComboBoxInteger (573,136 150x30), variable: GVL_Data.stRecipe.eLoadClose, text list: 'LineLoadClose'
    ComboBoxInteger (753,136 150x30), variable: GVL_Data.stRecipe.eProductType, text list: 'ProductType'
    Button (41,207 150x30), "手动下UC"
        toggle GVL.stSetting.bManualUnloadUc
    Button (219,207 150x30), "手动下工装"
        toggle GVL.stSetting.bManualUnloadFrock
    Button (1113,136 150x30), "手动上料"
        toggle GVL.stSetting.bManualLoad
    Button (397,207 150x30), "主流线分料屏蔽"
        toggle GVL.stSetting.bLine0BufferShield
    Button (573,207 150x30), "蜂鸣器屏蔽"
        toggle G_stSystem.stInput.bQuiet
    Button (753,207 150x30), "安全门屏蔽"
        toggle GVL.stSetting.bSafeDoorShield
    Button (933,207 150x30), "保压解除功能屏蔽"
        toggle GVL.stSetting.bOpenLockPressShield
    ComboBoxInteger (933,136 150x30), variable: GVL_Data.stRecipe.eLoadClass, text list: 'LineLoadClase'
    Button (41,278 150x30), "不允许前站放料"
        toggle GVL.stSetting.bStopFrontStation
    Button (1113,207 150x30), "工装误合盖检测屏蔽"
        toggle GVL.stSetting.bFrockCloseCheckShield
    RoundedRectangle (215,503 95x26), "%dms", text variable: GVL_Data.stRecipe.arrAutoTon[E_Timer.Line0PriorityOnDelay]
        OnMouseClick: write the text variable via Default
    Label (34,501 173x30), "主流线优先置位延时"
    RoundedRectangle (215,541 95x26), "%dms", text variable: GVL_Data.stRecipe.arrAutoTon[E_Timer.Line0PriorityOffDelay]
        OnMouseClick: write the text variable via Default
    Label (34,539 173x30), "主流线优先复位延时"
    Label (136,454 72x30), "共通"
    Label (458,453 72x30), "367机型"
    Line (336,466) (336,731)
    Line (666,466) (666,731)
    Label (787,453 72x30), "预留"
    Line (985,466) (985,731)
    Label (1134,452 72x30), "预留"
    RoundedRectangle (215,577 95x26), "%dms", text variable: GVL_Data.stRecipe.arrAutoTon[E_Timer.SteeringCheck1F]
        OnMouseClick: write the text variable via Default
    Label (34,575 173x30), "旋转站到位光电去抖动时间"
    RoundedRectangle (214,613 95x26), "%dms", text variable: GVL_Data.stRecipe.arrAutoTon[E_Timer.OpenLockCheckF]
        OnMouseClick: write the text variable via Default
    Label (33,611 173x30), "解锁站到位光电去抖动时间"
END_VISUALIZATION

// ---- VISUs/PageHome.TcVIS
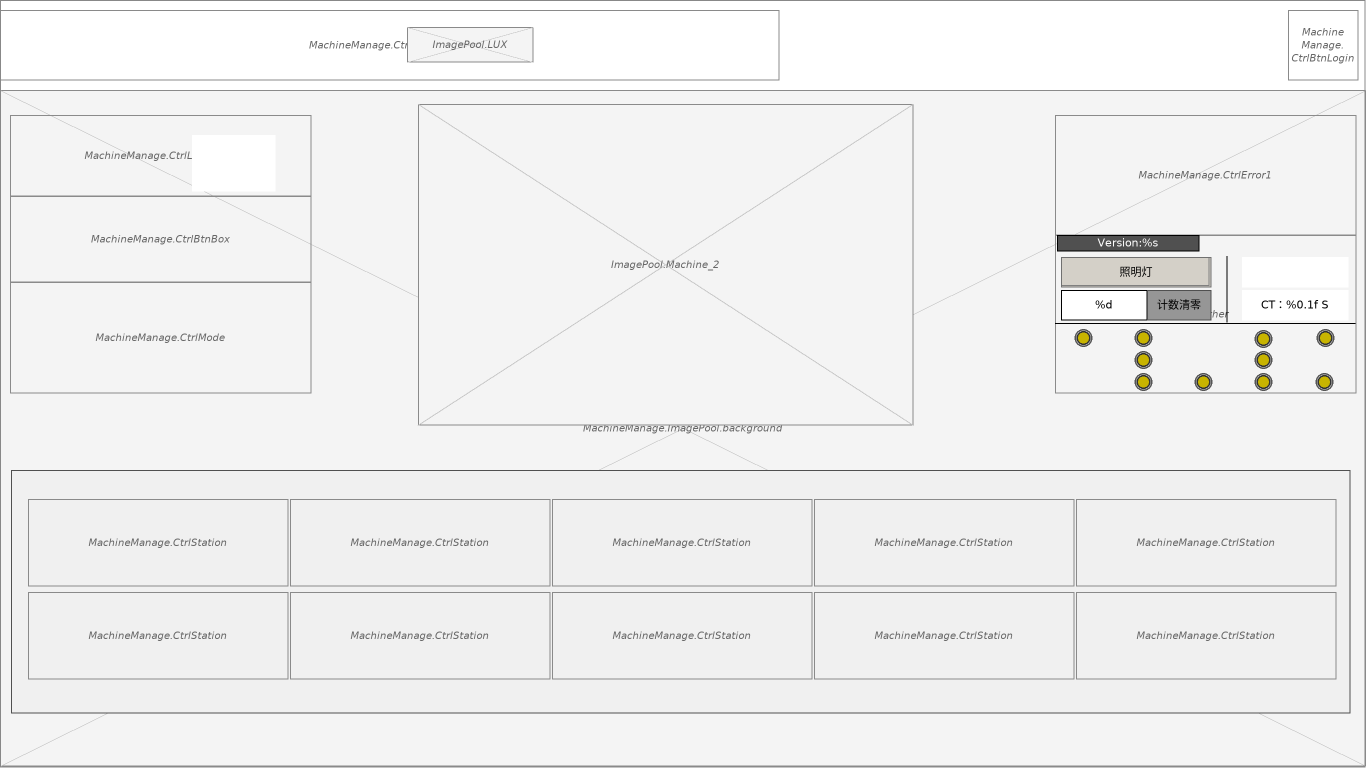
VISUALIZATION PageHome  // 1366x768
    Frame (0,0 1366x768)
        shows FrameMain()
    Frame (10,115 301x81)
        shows MachineManage.CtrlLanguage(System := G_stSystem)
    Frame (10,196 301x86)
        shows MachineManage.CtrlBtnBox(System := G_stSystem)
    Frame (10,282 301x111)
        shows MachineManage.CtrlMode(System := G_stSystem)
    Frame (1055,115 301x120)
        shows MachineManage.CtrlError1(System := G_stSystem, Error := G_stError.stNow)
    Frame (1055,235 301x158), text variable: P_System._fbCT.CycleTime
        shows CtrlOther()
    Rectangle (192,135 83x56)
    Button (1061,257 150x30), "照明灯"
        toggle GVL.Q.bLED
    Line (1227,322) (1227,256)
    Image (418,104 495x321), image: ImagePool.Machine_2
    Rectangle (1242,257 106x30), text list: 'MachineType', text index: GVL_Data.stRecipe.eMachineType
    Rectangle (1057,235 142x16), "Version:%s", text variable: MAIN.VERSION
    Rectangle (1242,290 106x30), "CT：%0.1f S", text variable: P_System._cttime
    Rectangle (1061,290 86x30), "%d", text variable: P_System._iProductionCount
    Rectangle (1147,290 64x30), "计数清零"
        tap P_System._bCountZero
    Lamp1 (1072,328 23x20), variable: GVL.I.bLine0Check2, style: Lamp-Lamp1-Yellow
    Line (1055,323) (1355,323)
    Lamp1 (1132,372 23x20), variable: GVL.I.bSteeringCheck1, style: Lamp-Lamp1-Yellow
    Lamp1 (1132,328 23x20), variable: GVL.I.bLine0Check3, style: Lamp-Lamp1-Yellow
    Lamp1 (1252,329 23x20), variable: GVL.I.bUnloadUcCheck2, style: Lamp-Lamp1-Yellow
    Lamp1 (1314,328 23x20), variable: GVL.I.bUnloadFrockConveyorCheck2, style: Lamp-Lamp1-Yellow
    Lamp1 (1192,372 23x20), variable: GVL.I.bOpenLockCheck, style: Lamp-Lamp1-Yellow
    Lamp1 (1252,372 23x20), variable: GVL.I.bTakeUcCheck1, style: Lamp-Lamp1-Yellow
    Lamp1 (1313,372 23x20), variable: GVL.I.bUnloadFrockCheck1, style: Lamp-Lamp1-Yellow
    Lamp1 (1132,350 23x20), variable: GVL.I.bAcquireCheck2, style: Lamp-Lamp1-Yellow
    Lamp1 (1252,350 23x20), variable: GVL.I.bUnloadUcCheck1, style: Lamp-Lamp1-Yellow
    Rectangle (11,470 1339x243)
    Frame (290,592 260x87)
        shows MachineManage.CtrlStation(System := G_stSystem, Station := G_arrStation[5])
    Frame (552,592 260x87)
        shows MachineManage.CtrlStation(System := G_stSystem, Station := G_arrStation[6])
    Frame (814,592 260x87)
        shows MachineManage.CtrlStation(System := G_stSystem, Station := G_arrStation[7])
    Frame (1076,592 260x87)
        shows MachineManage.CtrlStation(System := G_stSystem, Station := G_arrStation[8])
    Frame (1076,499 260x87)
        shows MachineManage.CtrlStation(System := G_stSystem, Station := G_arrStation[9])
    Frame (28,499 260x87)
        shows MachineManage.CtrlStation(System := G_stSystem, Station := G_arrStation[0])
    Frame (290,499 260x87)
        shows MachineManage.CtrlStation(System := G_stSystem, Station := G_arrStation[1])
    Frame (552,499 260x87)
        shows MachineManage.CtrlStation(System := G_stSystem, Station := G_arrStation[2])
    Frame (814,499 260x87)
        shows MachineManage.CtrlStation(System := G_stSystem, Station := G_arrStation[3])
    Frame (28,592 260x87)
        shows MachineManage.CtrlStation(System := G_stSystem, Station := G_arrStation[4])
END_VISUALIZATION

// ---- VISUs/PageMessage.TcVIS
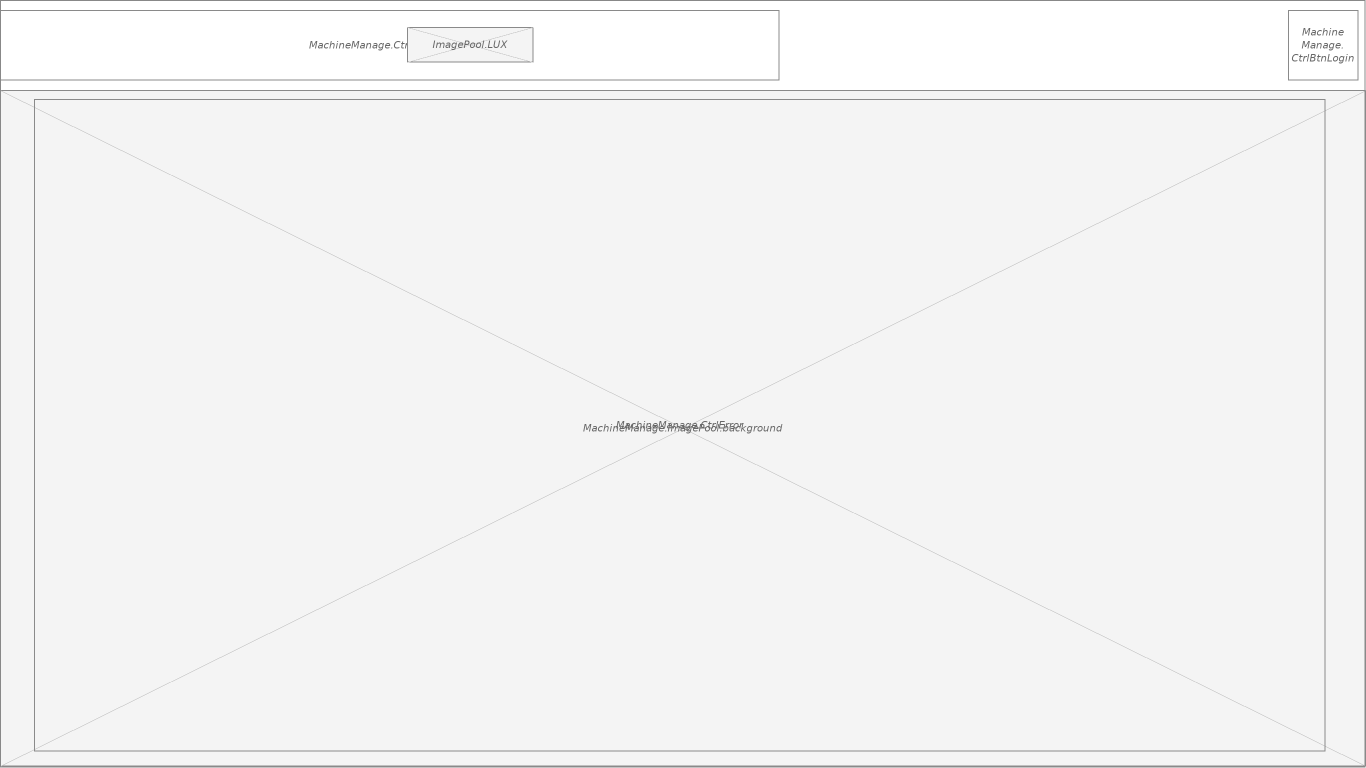
VISUALIZATION PageMessage  // 1366x768
    Frame (0,0 1366x768)
        shows FrameMain()
    Frame (34,99 1291x652)
        shows MachineManage.CtrlError(System := G_stSystem, Error := G_stError)
END_VISUALIZATION

// ---- VISUs/PageMonitor.TcVIS
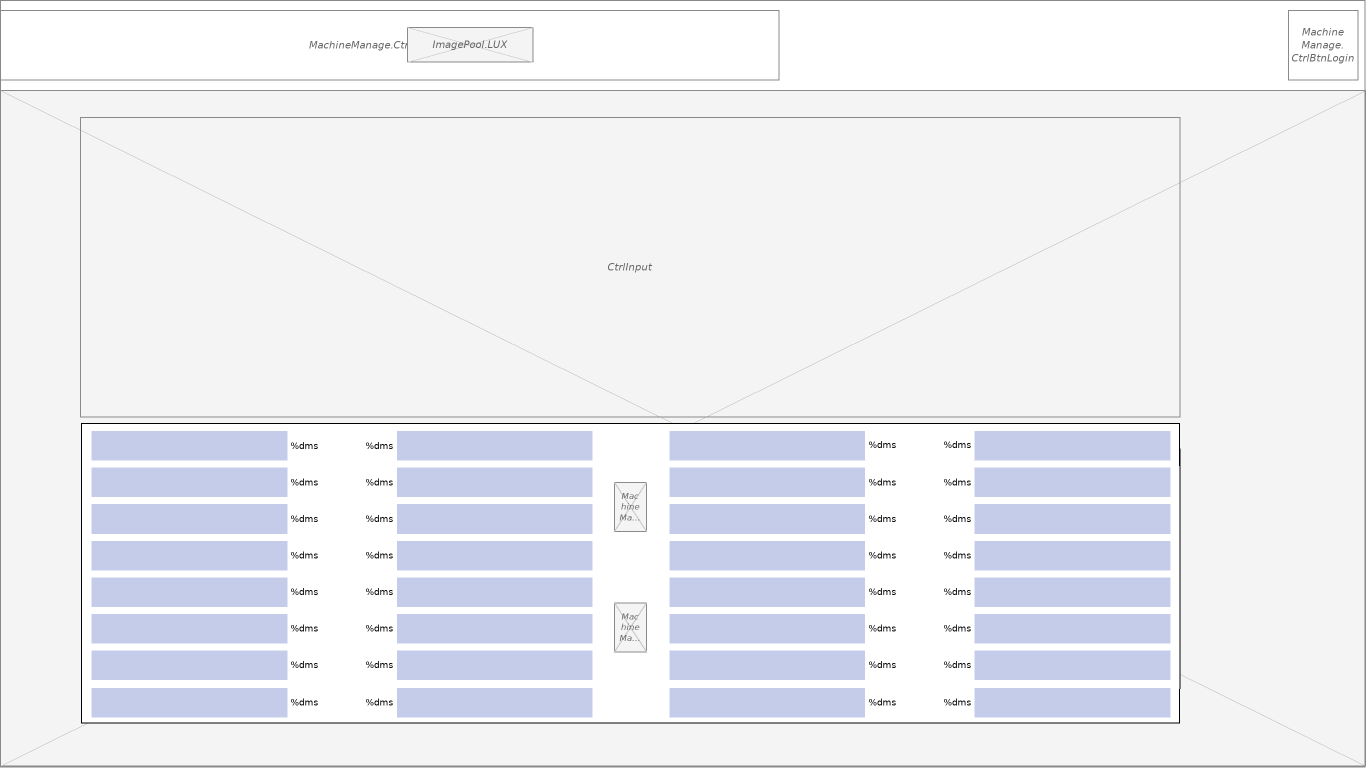
VISUALIZATION PageMonitor  // 1366x768
    Frame (0,0 1366x768)
        shows FrameMain()
    Frame (80,117 1100x300)
        shows CtrlInput(In := ADR(GVL_IO.I_Temp), SizeIn := Sizeof(GVL_IO.I_Temp), Enable := false, Ton := ADR(GVL_Data.stRecipe.arrInputTon), In_S := ADR(GVL.stShield_I))
    Frame (81,423 1100x300)
        shows CtrlOutput(In := ADR(GVL_IO.Q_Temp), SizeIn := sizeof(GVL_IO.Q_Temp), Enable := G_stSystem.stMode.bSetting, Ton := ADR(GVL_Data.stRecipe.arrOutputTon), In_S := ADR(GVL.stShield_Q))
END_VISUALIZATION

// ---- VISUs/PageSetting_AcquireLoad.TcVIS
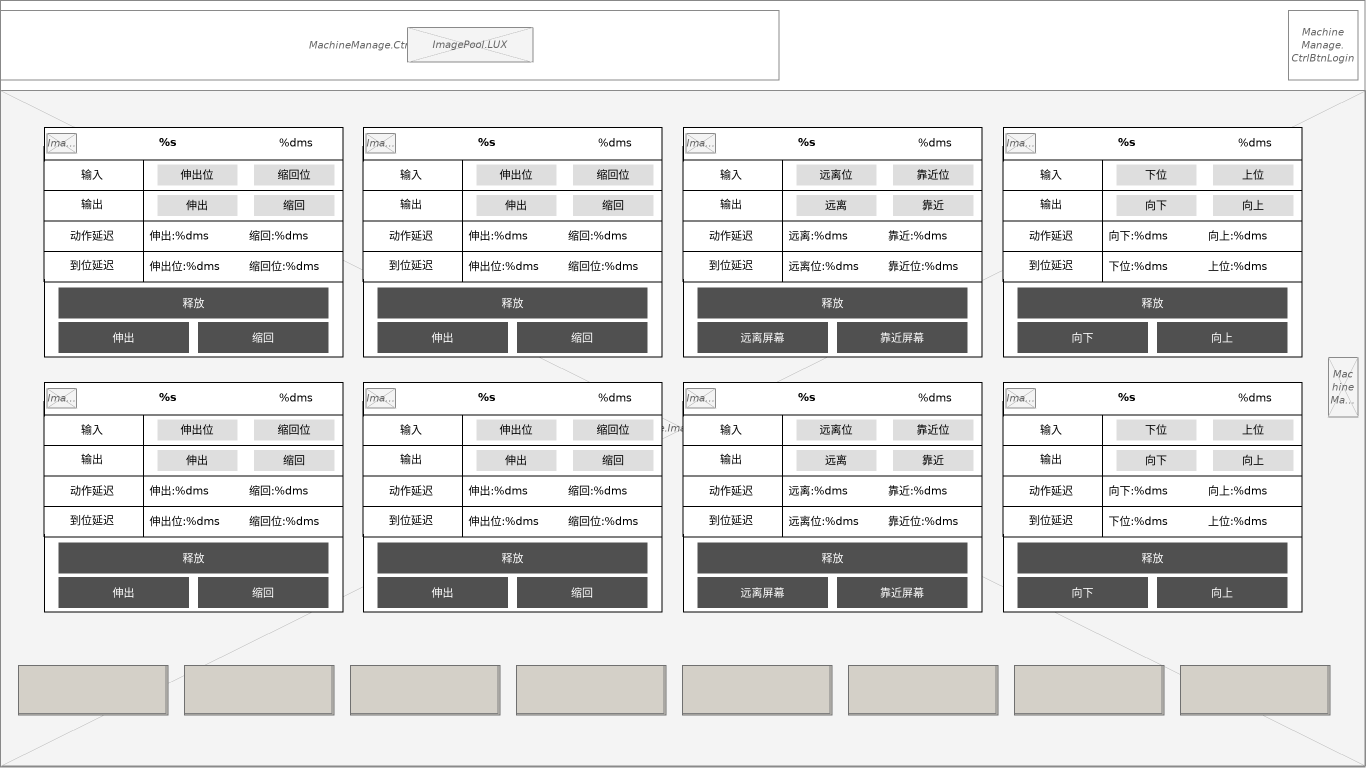
VISUALIZATION PageSetting_AcquireLoad  // 1366x768
    Frame (0,0 1366x768)
        shows CtrlPageSetting()
    Frame (45,127 300x230)
        shows Cyliner1(System := G_stSystem, Cylinder := G_arrCylinder[E_Cylinder.Line0Part], CylinderData := G_arrCylinderData[E_Cylinder.Line0Part])
    Frame (364,127 300x230)
        shows Cyliner1(System := G_stSystem, Cylinder := G_arrCylinder[E_Cylinder.Line0Prevent], CylinderData := G_arrCylinderData[E_Cylinder.Line0Prevent])
    Frame (45,382 300x230)
        shows Cyliner1(System := G_stSystem, Cylinder := G_arrCylinder[E_Cylinder.AcquirePrevent1], CylinderData := G_arrCylinderData[E_Cylinder.AcquirePrevent1])
    Frame (364,382 300x230)
        shows Cyliner1(System := G_stSystem, Cylinder := G_arrCylinder[E_Cylinder.AcquireLift], CylinderData := G_arrCylinderData[E_Cylinder.AcquireLift])
    Frame (683,382 300x230)
        shows Cyliner2(System := G_stSystem, Cylinder := G_arrCylinder[E_Cylinder.AcquirePush], CylinderData := G_arrCylinderData[E_Cylinder.AcquirePush])
    Frame (1003,382 300x230)
        shows Cyliner3(System := G_stSystem, Cylinder := G_arrCylinder[E_Cylinder.AcquireElevator], CylinderData := G_arrCylinderData[E_Cylinder.AcquireElevator])
    Frame (683,127 300x230)
        shows Cyliner2(System := G_stSystem, Cylinder := G_arrCylinder[E_Cylinder.Line0Push], CylinderData := G_arrCylinderData[E_Cylinder.Line0Push])
    Image (1328,357 30x60), image: MachineManage.ImagePool.next
        OnMouseClick: change screen: PageSetting_AcquireLoad_2
    Frame (1003,127 300x230)
        shows Cyliner3(System := G_stSystem, Cylinder := G_arrCylinder[E_Cylinder.Line0PushElevator], CylinderData := G_arrCylinderData[E_Cylinder.Line0PushElevator])
END_VISUALIZATION

// ---- VISUs/PageSetting_AcquireLoad_2.TcVIS
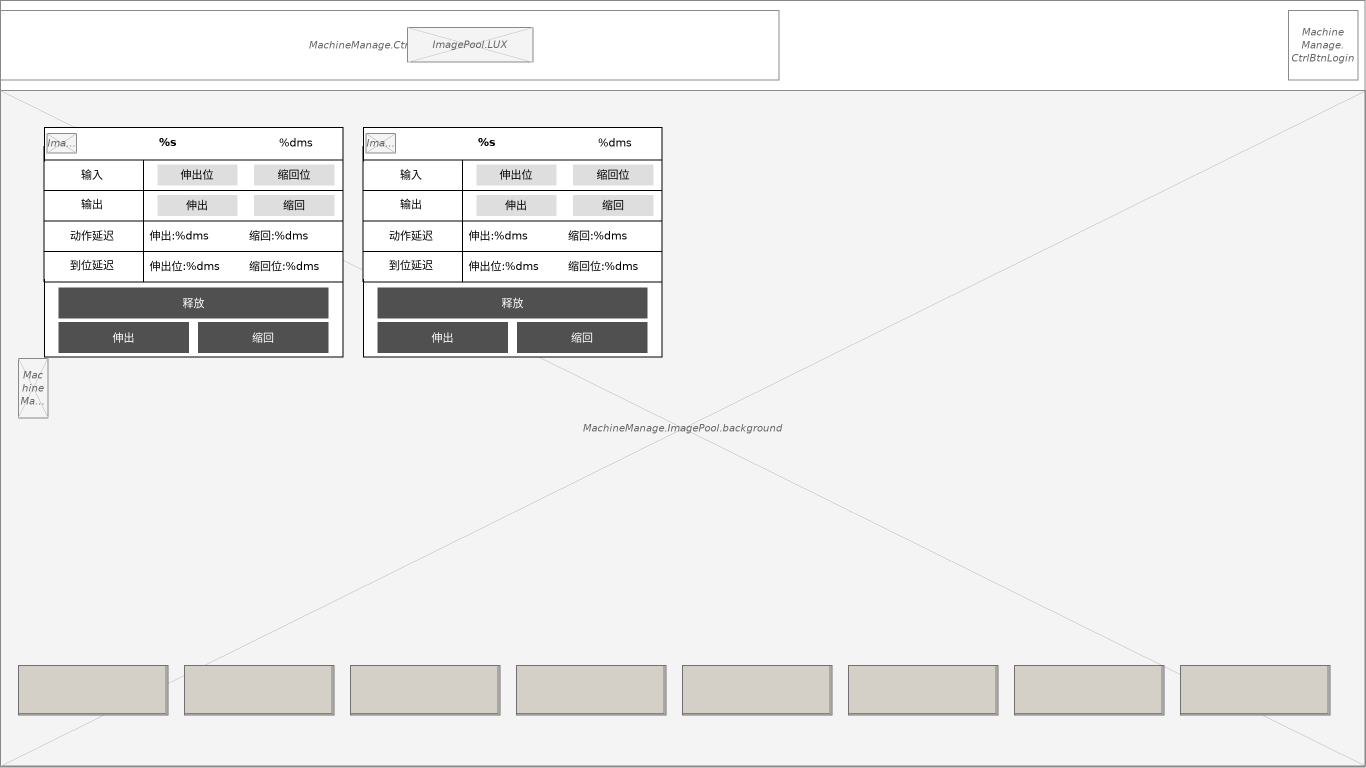
VISUALIZATION PageSetting_AcquireLoad_2  // 1366x768
    Frame (0,0 1366x768)
        shows CtrlPageSetting()
    Frame (45,127 300x230)
        shows Cyliner1(System := G_stSystem, Cylinder := G_arrCylinder[E_Cylinder.AcquirePrevent2], CylinderData := G_arrCylinderData[E_Cylinder.AcquirePrevent2])
    Image (18,358 30x60), image: MachineManage.ImagePool.prev
        OnMouseClick: change screen: PageSetting_AcquireLoad
    Frame (364,127 300x230)
        shows Cyliner1(System := G_stSystem, Cylinder := G_arrCylinder[E_Cylinder.AcquirePrevent0], CylinderData := G_arrCylinderData[E_Cylinder.AcquirePrevent0])
END_VISUALIZATION

// ---- VISUs/PageSetting_OpenLock_2.TcVIS
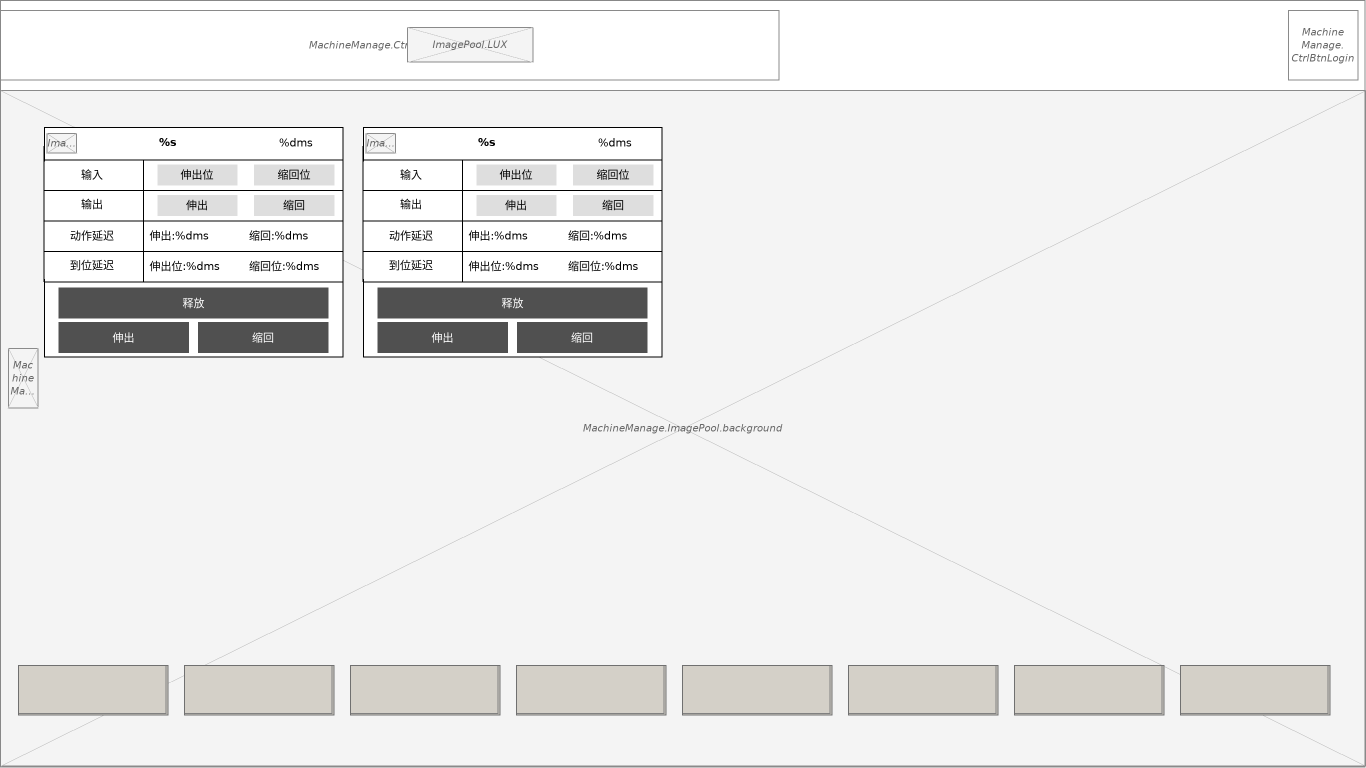
VISUALIZATION PageSetting_OpenLock_2  // 1366x768
    Frame (0,0 1366x768)
        shows CtrlPageSetting()
    Frame (45,127 300x230)
        shows Cyliner1(System := G_stSystem, Cylinder := G_arrCylinder[E_Cylinder.OpenLockPressPush], CylinderData := G_arrCylinderData[E_Cylinder.OpenLockPressPush])
    Frame (364,127 300x230)
        shows Cyliner1(System := G_stSystem, Cylinder := G_arrCylinder[E_Cylinder.OpenLockPressRotate], CylinderData := G_arrCylinderData[E_Cylinder.OpenLockPressRotate])
    Image (8,348 30x60), image: MachineManage.ImagePool.prev
        OnMouseClick: change screen: PageSetting_OpenLock
END_VISUALIZATION

// ---- VISUs/PageSetting_TakeUc.TcVIS
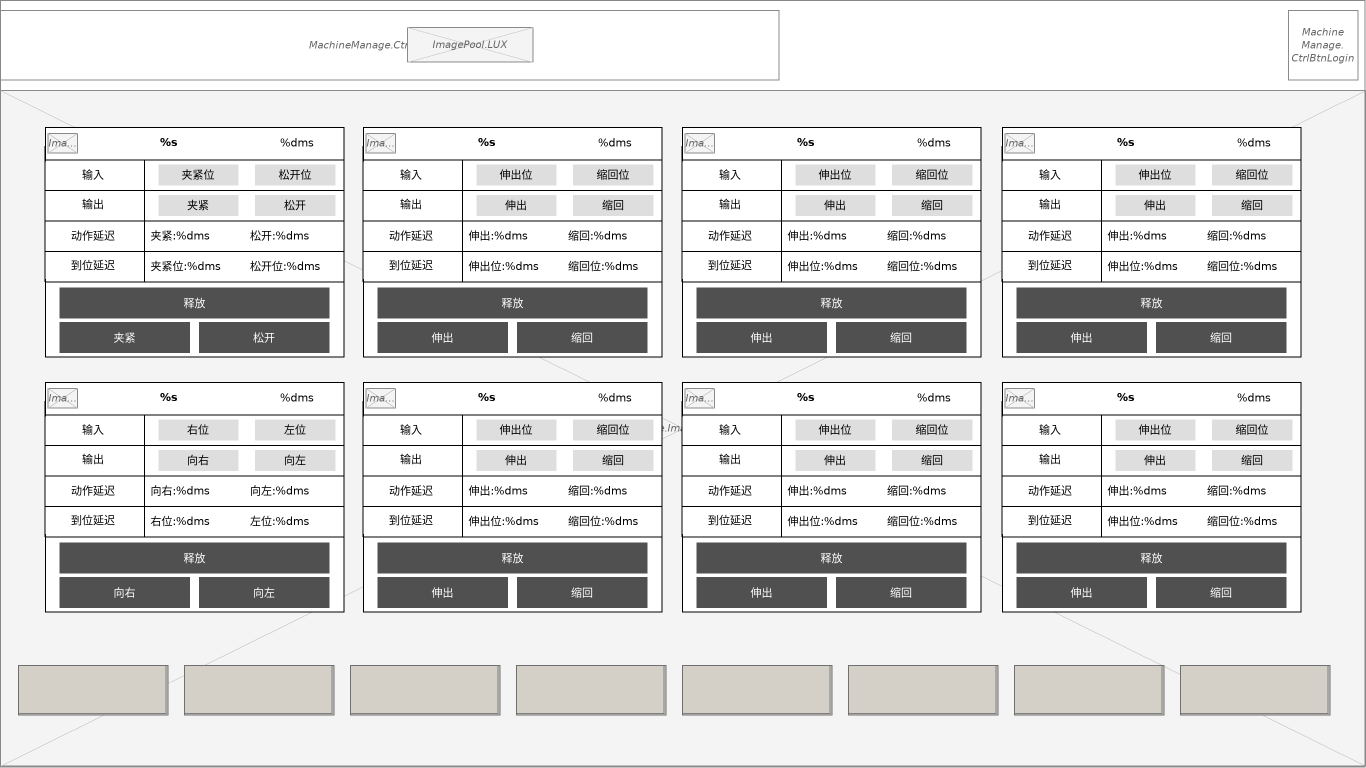
VISUALIZATION PageSetting_TakeUc  // 1366x768
    Frame (0,0 1366x768)
        shows CtrlPageSetting()
    Frame (364,127 300x230)
        shows Cyliner1(System := G_stSystem, Cylinder := G_arrCylinder[E_Cylinder.TakeUcPrevent], CylinderData := G_arrCylinderData[E_Cylinder.TakeUcPrevent])
    Frame (683,127 300x230)
        shows Cyliner1(System := G_stSystem, Cylinder := G_arrCylinder[E_Cylinder.TakeUcLift], CylinderData := G_arrCylinderData[E_Cylinder.TakeUcLift])
    Frame (1003,127 300x230)
        shows Cyliner1(System := G_stSystem, Cylinder := G_arrCylinder[E_Cylinder.TakeUcPush], CylinderData := G_arrCylinderData[E_Cylinder.TakeUcPush])
    Frame (45,382 300x230)
        shows Cyliner4(System := G_stSystem, Cylinder := G_arrCylinder[E_Cylinder.TakeUcRotate], CylinderData := G_arrCylinderData[E_Cylinder.TakeUcRotate])
    Frame (364,382 300x230)
        shows Cyliner1(System := G_stSystem, Cylinder := G_arrCylinder[E_Cylinder.TakeUcStandard], CylinderData := G_arrCylinderData[E_Cylinder.TakeUcStandard])
    Frame (683,382 300x230)
        shows Cyliner1(System := G_stSystem, Cylinder := G_arrCylinder[E_Cylinder.TakeUcElevator], CylinderData := G_arrCylinderData[E_Cylinder.TakeUcElevator])
    Frame (1003,382 300x230)
        shows Cyliner1(System := G_stSystem, Cylinder := G_arrCylinder[E_Cylinder.TakeUcPush1], CylinderData := G_arrCylinderData[E_Cylinder.TakeUcPush1])
    Frame (45,127 300x230)
        shows Cyliner5(System := G_stSystem, Cylinder := G_arrCylinder[E_Cylinder.TakeUcFrockClamp], CylinderData := G_arrCylinderData[E_Cylinder.TakeUcFrockClamp])
END_VISUALIZATION

// ---- VISUs/PageSetting_Steering.TcVIS
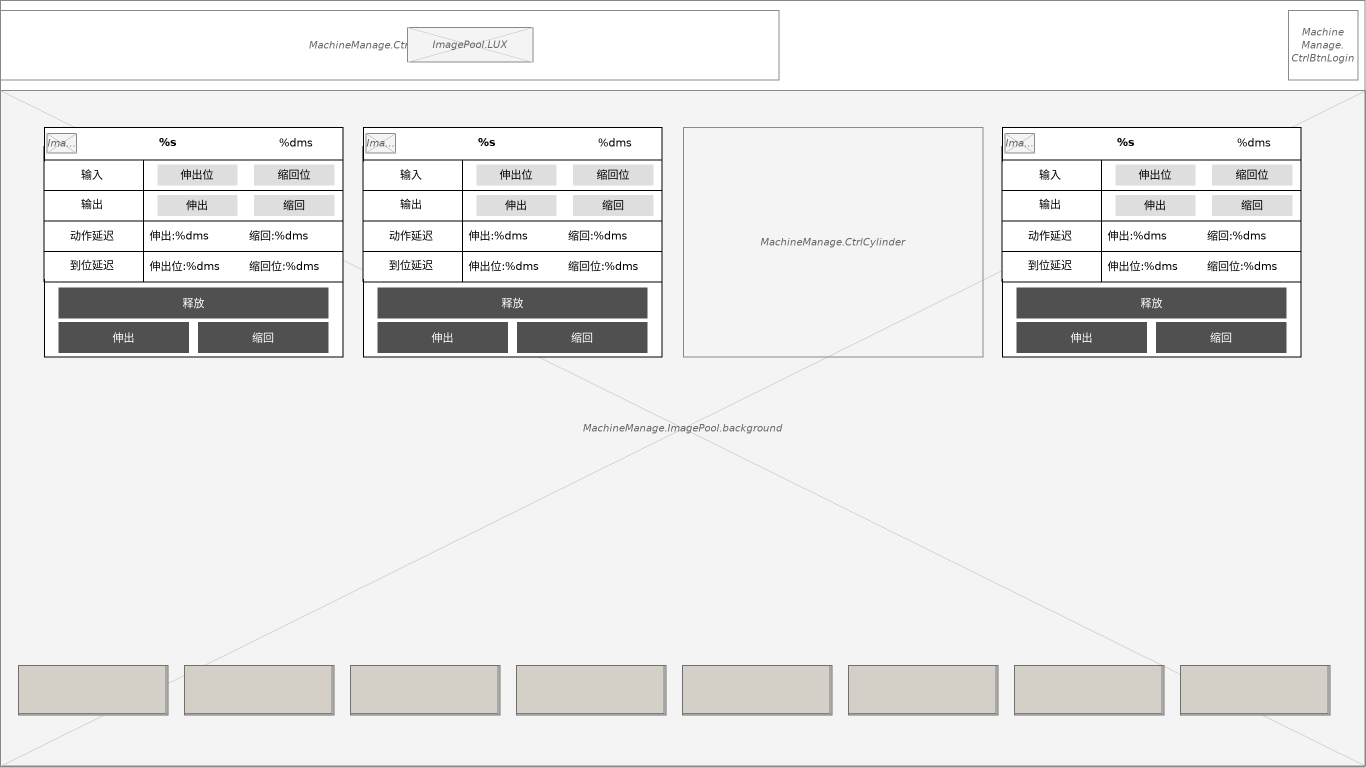
VISUALIZATION PageSetting_Steering  // 1366x768
    Frame (0,0 1366x768)
        shows CtrlPageSetting()
    Frame (45,127 300x230)
        shows Cyliner1(System := G_stSystem, Cylinder := G_arrCylinder[E_Cylinder.SteeringLift], CylinderData := G_arrCylinderData[E_Cylinder.SteeringLift])
    Frame (364,127 300x230)
        shows Cyliner1(System := G_stSystem, Cylinder := G_arrCylinder[E_Cylinder.SteeringAcquireElevator], CylinderData := G_arrCylinderData[E_Cylinder.SteeringAcquireElevator])
    Frame (683,127 300x230)
        shows MachineManage.CtrlCylinder(System := G_stSystem, Cylinder := G_arrCylinder[E_Cylinder.SteeringRotate], CylinderData := G_arrCylinderData[E_Cylinder.SteeringRotate])
    Frame (1003,127 300x230)
        shows Cyliner1(System := G_stSystem, Cylinder := G_arrCylinder[E_Cylinder.SteeringAcquireLimit], CylinderData := G_arrCylinderData[E_Cylinder.SteeringAcquireLimit])
END_VISUALIZATION

// ---- VISUs/PageSetting_Other.TcVIS
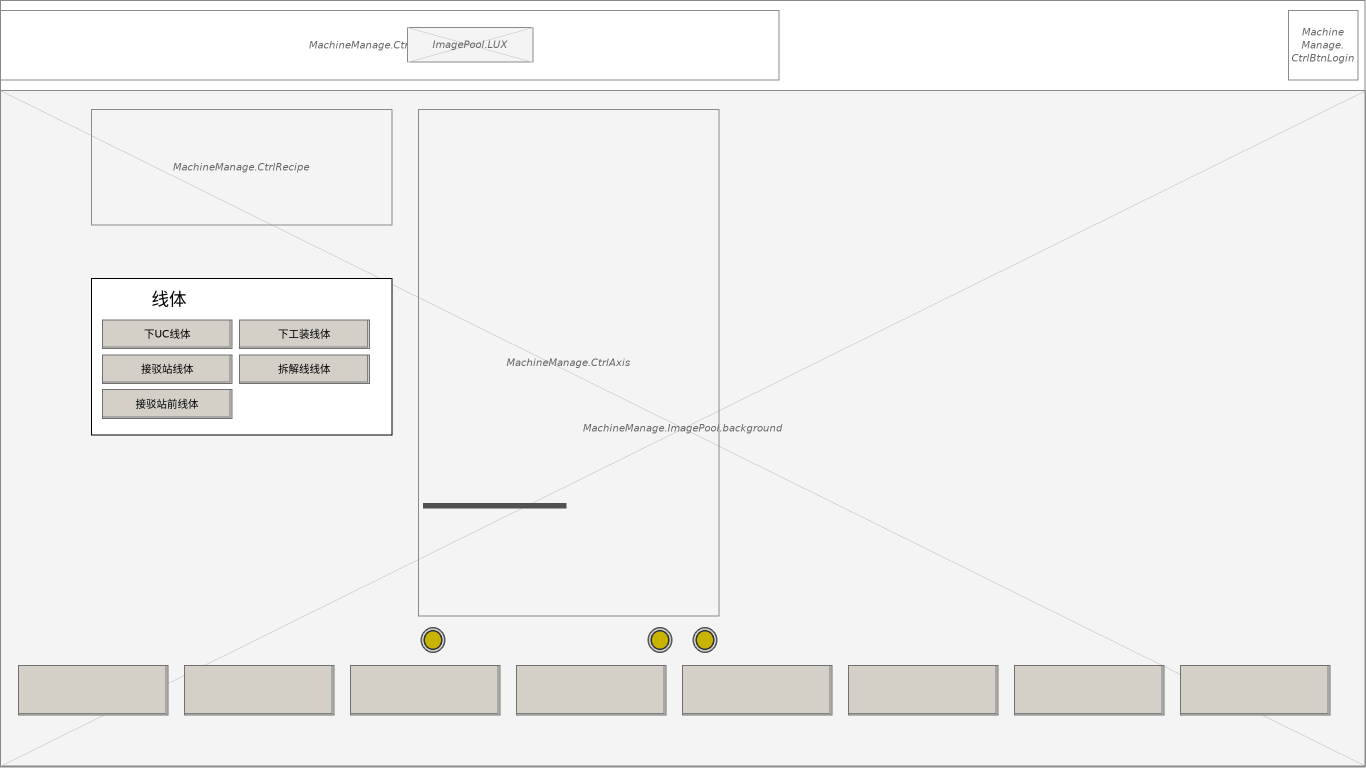
VISUALIZATION PageSetting_Other  // 1366x768
    Frame (0,0 1366x768)
        shows CtrlPageSetting()
    Frame (418,109 301x507)
        shows MachineManage.CtrlAxis(System := G_stSystem, Axis := G_arrAxis[E_Axis.Z], Data := G_arrAxisData[E_Axis.Z])
    Frame (419,625 300x30)
        shows CtrlAxisInput(In := GVL_IO.AxisInput)
    Frame (91,109 301x116)
        shows MachineManage.CtrlRecipe()
    Frame (91,278 301x157)
        shows CtrlLine()
    Rectangle (423,503 143x5), colour toggle: G_arrAxis[E_Axis.Z].Axis_REF.Status.Error OR G_arrAxis[E_Axis.Z].Axis_REF.Status.Disabled
END_VISUALIZATION

// ---- VISUs/PageSetting_Unload_L.TcVIS
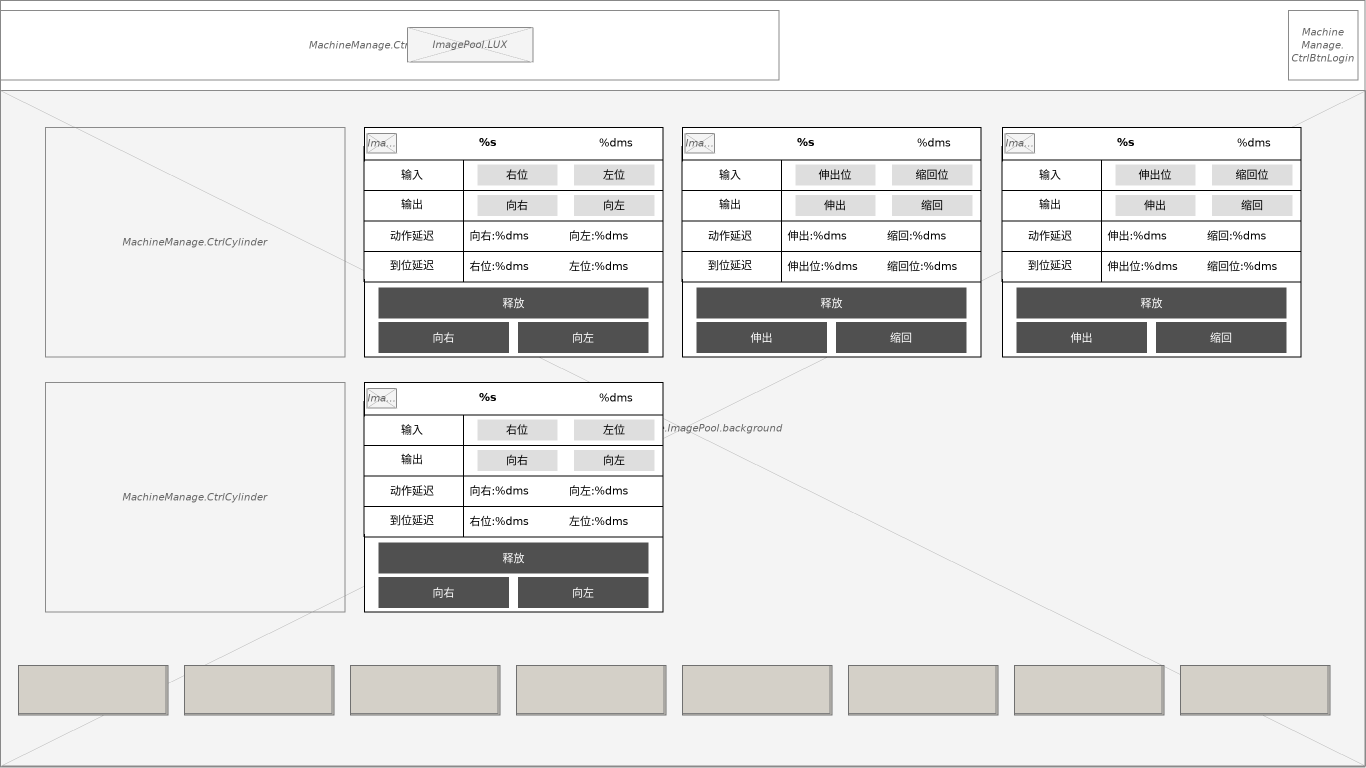
VISUALIZATION PageSetting_Unload_L  // 1366x768
    Frame (0,0 1366x768)
        shows CtrlPageSetting()
    Frame (683,127 300x230)
        shows Cyliner1(System := G_stSystem, Cylinder := G_arrCylinder[E_Cylinder.UnloadUcBeltTipper], CylinderData := G_arrCylinderData[E_Cylinder.UnloadUcBeltTipper])
    Frame (1003,127 300x230)
        shows Cyliner1(System := G_stSystem, Cylinder := G_arrCylinder[E_Cylinder.UnloadUcBeltLift], CylinderData := G_arrCylinderData[E_Cylinder.UnloadUcBeltLift])
    Frame (45,127 300x230)
        shows MachineManage.CtrlCylinder(System := G_stSystem, Cylinder := G_arrCylinder[E_Cylinder.UnloadFrockConveyorPrevent], CylinderData := G_arrCylinderData[E_Cylinder.UnloadFrockConveyorPrevent])
    Frame (364,127 300x230)
        shows Cyliner4(System := G_stSystem, Cylinder := G_arrCylinder[E_Cylinder.UnloadFrockConveyorPush], CylinderData := G_arrCylinderData[E_Cylinder.UnloadFrockConveyorPush])
    Frame (45,382 300x230)
        shows MachineManage.CtrlCylinder(System := G_stSystem, Cylinder := G_arrCylinder[E_Cylinder.UnloadUcElevator], CylinderData := G_arrCylinderData[E_Cylinder.UnloadUcElevator])
    Frame (364,382 300x230)
        shows Cyliner4(System := G_stSystem, Cylinder := G_arrCylinder[E_Cylinder.UnloadUcConveyorPush], CylinderData := G_arrCylinderData[E_Cylinder.UnloadUcConveyorPush])
END_VISUALIZATION

